: REAL; arScrew[98].rWidth : REAL; arScrew[98].rAngle_knives : REAL; arScrew[98].rMidle_line : REAL; arScrew[98].rInstal_support : REAL; arScrew[98].rPosX0 : REAL; arScrew[98].rPosX1 : REAL; arScrew[98].rPosX2 : REAL; arScrew[98].equip.place : WSTRING(10); arScrew[98].equip.name : WSTRING(20); arScrew[98].name : WSTRING(20); arScrew[99].rRstmax : REAL; arScrew[99].rRstmin : REAL; arScrew[99].iCountCycle : INT; arScrew[99].iActuatorsMove : INT; arScrew[99].iActuatorsStep : INT; arScrew[99].iActuatorsStartPos[0] : INT; arScrew[99].iActuatorsStartPos[1] : INT; arScrew[99].support[0].bPosition : BOOL; arScrew[99].support[0].arLength[0] : INT; arScrew[99].support[0].arLength[1] : INT; arScrew[99].support[0].name : WSTRING(20); arScrew[99].support[1].bPosition : BOOL; arScrew[99].support[1].arLength[0] : INT; arScrew[99].support[1].arLength[1] : INT; arScrew[99].support[1].name : WSTRING(20); arScrew[99].bDirRotate : BOOL; arScrew[99].rOut_diam : REAL; arScrew[99].rInner_diam : REAL; arScrew[99].rTurn_step : REAL; arScrew[99].rWidth : REAL; arScrew[99].rAngle_knives : REAL; arScrew[99].rMidle_line : REAL; arScrew[99].rInstal_support : REAL; arScrew[99].rPosX0 : REAL; arScrew[99].rPosX1 : REAL; arScrew[99].rPosX2 : REAL; arScrew[99].equip.place : WSTRING(10); arScrew[99].equip.name : WSTRING(20); arScrew[99].name : WSTRING(20); arScrew[100].rRstmax : REAL; arScrew[100].rRstmin : REAL; arScrew[100].iCountCycle : INT; arScrew[100].iActuatorsMove : INT; arScrew[100].iActuatorsStep : INT; arScrew[100].iActuatorsStartPos[0] : INT; arScrew[100].iActuatorsStartPos[1] : INT; arScrew[100].support[0].bPosition : BOOL; arScrew[100].support[0].arLength[0] : INT; arScrew[100].support[0].arLength[1] : INT; arScrew[100].support[0].name : WSTRING(20); arScrew[100].support[1].bPosition : BOOL; arScrew[100].support[1].arLength[0] : INT; arScrew[100].support[1].arLength[1] : INT; arScrew[100].support[1].name : WSTRING(20); arScrew[100].bDirRotate : BOOL; arScrew[100].rOut_diam : REAL; arScrew[100].rInner_diam : REAL; arScrew[100].rTurn_step : REAL; arScrew[100].rWidth : REAL; arScrew[100].rAngle_knives : REAL; arScrew[100].rMidle_line : REAL; arScrew[100].rInstal_support : REAL; arScrew[100].rPosX0 : REAL; arScrew[100].rPosX1 : REAL; arScrew[100].rPosX2 : REAL; arScrew[100].equip.place : WSTRING(10); arScrew[100].equip.name : WSTRING(20); arScrew[100].name : WSTRING(20)
      global variables Global_Variables
      Vizualization/
        TextList/
          text list OnOffList
          text list MbBoud
          text list NoYes
          text list ModeSysList
          text list typeEquip
          text list Direction
          text list MbParity
          text list MbStopbit
          text list TypeSetup
          text list DirectRotation
        image pool Images
        visualisation Waiting
        ImagesPool/
          image pool sensPool
          image pool PumpPool
          image pool ValvePool
        7_inch/
          visualisation _Actuators
          visualisation _SettingsEquipment
          visualisation _Diag_geomtry_rec
          visualisation _Support
          visualisation _Equipment_2
          visualisation _Equipment_3
          visualisation _Diag_WARNING
          visualisation _TypeMachine
          visualisation _Diag_support_rec
          visualisation _Equip_7inch
          visualisation _Equipment_4
          visualisation _Diag_save
          visualisation _Equipment_1
          visualisation _Diag_geomtry_work
          visualisation _Steel_7inch
          visualisation _SettingsSens_7inch
          visualisation _Alarms_7inch
          visualisation _MAIN_7inch
          visualisation _Equipment
          visualisation _Recipe_7inch
          visualisation _Diag_ok
          visualisation _SettingsActuators
          visualisation _Diag_equip
          visualisation _SettingsMain_7inch
          visualisation _TimeSetup_7inch
          visualisation _Diag_supKey
      Alarm Configuration
        alarm group AlarmGroup
            8 [Error]: Comparison Equal, ExpressionToCompare    TRUE, Expression Actuators.bDr1_error - "Ошибка драйвера актуатора 1"
            9 [Error]: Comparison Equal, ExpressionToCompare TRUE, Expression Actuators.bDr2_error - "Ошибка драйвера актуатора 2"
            1 [Error]: Comparison Equal, ExpressionToCompare TRUE, Expression Main.fbKkMotor.bOUT - "Сработало тепловое реле элекродвигателя маслостанции"
            3 [Error]: Comparison Equal, ExpressionToCompare TRUE, Expression Main.fbControl.bAlarm - "Ошибка дижения рабочего цилиндра"
            4 [Error]: Comparison Equal, ExpressionToCompare TRUE, Expression Main.fbTimeMotor.bService - "Проведите плановое плановое ТО"
            5 [Error]: Comparison Equal, ExpressionToCompare TRUE, Expression Main.bSnsH - "Достигнута максимально крайняя точка движения (координата X4)"
            6 [Error]: Comparison Equal, ExpressionToCompare TRUE, Expression Main.bSnsL - "Достигнута минимально крайняя точка движения (координата X3)"
            7 [Error]: Comparison Equal, ExpressionToCompare TRUE, Expression Main.bNoConnect - "Нет сигнала с модулем ПР"
        alarm group WarningGroup
            0 [Warning]: Comparison Equal, ExpressionToCompare TRUE, Expression warn.bStartPos - "Начальная позиция актуаторов выходит за допустимы предел"
            1 [Warning]: Comparison Equal, ExpressionToCompare TRUE, Expression warn.bMaxMove - "Расчитанных ход актуаторов больше, чем их возможный"
            2 [Warning]: Comparison Equal, ExpressionToCompare TRUE, Expression warn.bNotSupport - "Нет подходящей поддержки"
        AlarmStorage
        alarm class Error (priority 10, acknowledge REP)
        text list AlarmGroup
        text list WarningGroup
        alarm class Warning (priority 11, acknowledge REP)
    Debug : Debug, Production association OWEN, version 3.5.17.3001 (disabled)
        unmapped channels: RAM used, RAM free, Open files, Processor usage, Core temp, Enable Debug, Debug pause
    Info : Info, Production association OWEN, version 3.5.17.3001 (disabled)
        unmapped channels: VENDOR, DEVICE, SERIAL, RUNTIME, FIRMWARE, LINUX, TARGET, PROJECT, AUTHOR, VERSION, PROFILE, LASTCHANGES
    OwenRTC : OwenRTC, Production association OWEN, version 3.5.17.3001 (disabled)
        unmapped channels: Year, Month, Day, Hour, Minute, Second, Day of Week, Week of Year, Format Date, Format Time, UTC Offset, NTP Enabled, NTP Error, System Timer, Date And Time, Operating Time, New Year, New Month, New Day, New Hour, New Minute, New Second, New UTC Offset, Set Settings DT, Enable NTP, Prefer Server
    OwenCloud : OwenCloud, Production association OWEN, version 3.5.17.3001 (disabled)
        unmapped channels: OwenCloud enabled, Folder error, Symbol error, No Symbol Config, Status, Enable OwenCloud
    Buzzer : Buzzer, Production association OWEN, version 3.5.17.3001 (disabled)
        unmapped channels: Buzzer enabled, Enable Buzzer, Sound frequency
    Watchdog : Watchdog, Production association OWEN, version 3.5.17.3001 (disabled)
        unmapped channels: Exception Handling, Last Exception Code, Last Exception Description, Last Exception Time, Hardware Watchdog Flag, Power Reboot Count, Watchdog Reboot Count, Exception Reboot Count, Command Reboot Count, Reboot, Reset Counters
    Drives : Drives, Production association OWEN, version 3.5.17.3001 (disabled)
        unmapped channels: FS size, FS used, FS free, USB Mounted, USB Unmount done, USB size, USB used, USB free, MMC Mounted, MMC Unmount done, MMC size, MMC used, MMC free, FS wear, Enable Drives, USB Unmount, MMC Unmount
    Screen : Screen, Production association OWEN, version 3.5.17.3001 (disabled)
        unmapped channels: Get Brightness, Dim time, Off time, Full brightness, Dim brightness, Off brightness, Dim visu name, Off visu name, On visu name, Wake up
    Network : Network, Production association OWEN, version 3.5.17.3001 (disabled)
        unmapped channels: DHCP enabled, IP, Mask, Gateway, MAC, Hostname, Enable DHCP, New IP, New Mask, New Gateway, New Hostname, Set Settings
    Modbus_COM : Modbus COM, 3S - Smart Software Solutions GmbH, version 3.5.16.0
        settings: DataBits = 8; StopBits = 1; ComPort = 1
      Modbus_Master_COM_Port : Modbus Master, COM Port, 3S - Smart Software Solutions GmbH, version 3.5.17.0
          settings: Transmission = 'RTU'; ResponseTimeout = 50; TimeBetweenFrames = 30; Auto-restart communication = TRUE
        AI_module : Modbus Slave, COM Port, 3S - Smart Software Solutions GmbH, version 3.5.16.0
            settings: SlaveAddress = 16; ResponseTimeout = 20; UseExtendedFunctionCodes = TRUE; Channel 0.Function Code = 3; Channel 0.Read Offset = 16#0200; Channel 0.Read Length = 7; Channel 0.Write Offset = 0; Channel 0.Write Length = 0; Channel 0.Cycle Time = 20; Channel 1.Function Code = 16; Channel 1.Read Offset = 0; Channel 1.Read Length = 0; Channel 1.Write Offset = 16#0214; Channel 1.Write Length = 11; Channel 1.Cycle Time = 20; Channel 3.Function Code = 16; Channel 3.Read Offset = 0; Channel 3.Read Length = 0; Channel 3.Write Offset = 16#021F; Channel 3.Write Length = 4; Channel 3.Cycle Time = 20; Channel 4.Function Code = 3; Channel 4.Read Offset = 16#0207; Channel 4.Read Length = 3; Channel 4.Write Offset = 0; Channel 4.Write Length = 0; Channel 4.Cycle Time = 20
            input  inArWord : ARRAY[0..6] OF WORD  // Channel 0
            input  readSec : WORD  // Channel 0.Channel 0
            input  DI1 : WORD  // Channel 0.Channel 0
            input  DO1 : WORD  // Channel 0.Channel 0
            output writeX0 : WORD  // Channel 1.Channel 1
            output writeX1 : WORD  // Channel 1.Channel 1
            output writeX2 : WORD  // Channel 1.Channel 1
            output writeX3 : WORD  // Channel 1.Channel 1
            output writeX4 : WORD  // Channel 1.Channel 1
            output writeSec : WORD  // Channel 1.Channel 1
            output writeMode : WORD  // Channel 1.Channel 1
            output writeData : WORD  // Channel 1.Channel 1
            output writeMinL : WORD  // Channel 1.Channel 1
            output writeMaxL : WORD  // Channel 1.Channel 1
            output writeOffset : WORD  // Channel 1.Channel 1
            output writeImpMaxDr1 : WORD  // Channel 3.Channel 3
            output writeImpMaxDr2 : WORD  // Channel 3.Channel 3
            output writeImpSetpDr1 : WORD  // Channel 3.Channel 3
            output writeImpSetpDr2 : WORD  // Channel 3.Channel 3
            input  readStateDr : WORD  // Channel 4.Channel 4
            input  readCntImpDr1 : WORD  // Channel 4.Channel 4
            input  readCntImpDr2 : WORD  // Channel 4.Channel 4
            unmapped channels: Channel 1, Channel 3, Channel 4
  5ce3da45-db07-42e7-a21c-a00fff4ed8f6|D:\png для cWeb\KSp_alarm.png
  5ce3da45-db07-42e7-a21c-a00fff4ed8f6|D:\png для cWeb\SU_on.png
  5ce3da45-db07-42e7-a21c-a00fff4ed8f6|D:\png для cWeb\SU_off.png
  5ce3da45-db07-42e7-a21c-a00fff4ed8f6|background.jpeg
  5ce3da45-db07-42e7-a21c-a00fff4ed8f6|D:\png для cWeb\TO_SPAD.png
  5ce3da45-db07-42e7-a21c-a00fff4ed8f6|D:\png для cWeb\FO_alarm.png
  5ce3da45-db07-42e7-a21c-a00fff4ed8f6|background1.jpg
  5ce3da45-db07-42e7-a21c-a00fff4ed8f6|C:\Users\Андрей\Downloads\background_SuUP.jpg
  5ce3da45-db07-42e7-a21c-a00fff4ed8f6|C:\Users\Андрей\Downloads\лого1.png
  5ce3da45-db07-42e7-a21c-a00fff4ed8f6|C:\Users\Андрей\Downloads\background_FoDW.jpg
  5ce3da45-db07-42e7-a21c-a00fff4ed8f6|D:\png для cWeb\EK_on.png
  5ce3da45-db07-42e7-a21c-a00fff4ed8f6|C:\Users\Андрей\Downloads\miniLogo_white.png
  5ce3da45-db07-42e7-a21c-a00fff4ed8f6|C:\Users\Андрей\Downloads\background_FanUP.jpg
  5ce3da45-db07-42e7-a21c-a00fff4ed8f6|D:\png для cWeb\TO_freeze.png
  5ce3da45-db07-42e7-a21c-a00fff4ed8f6|D:\png для cWeb\DumpIn_off_op.png
  5ce3da45-db07-42e7-a21c-a00fff4ed8f6|D:\png для cWeb\EK_alarm.png
  5ce3da45-db07-42e7-a21c-a00fff4ed8f6|D:\png для cWeb\Pump_left_alarm.png
  5ce3da45-db07-42e7-a21c-a00fff4ed8f6|D:\png для cWeb\Fan_right_on.png
  5ce3da45-db07-42e7-a21c-a00fff4ed8f6|C:\Users\Андрей\Downloads\background_GenUP.jpg
  5ce3da45-db07-42e7-a21c-a00fff4ed8f6|D:\png для cWeb\SU_alarm.png
  5ce3da45-db07-42e7-a21c-a00fff4ed8f6|C:\Users\Андрей\Downloads\background_SuDW.jpg
  5ce3da45-db07-42e7-a21c-a00fff4ed8f6|D:\Program's\картинки для мнемосхем\svg\Arrow_Black_Left.svg
  5ce3da45-db07-42e7-a21c-a00fff4ed8f6|D:\png для cWeb\Filter_Alarm.png
  5ce3da45-db07-42e7-a21c-a00fff4ed8f6|D:\png для cWeb\KSp_off.png
  5ce3da45-db07-42e7-a21c-a00fff4ed8f6|D:\Program's\картинки для мнемосхем\Избранные\Warning.png
  5ce3da45-db07-42e7-a21c-a00fff4ed8f6|D:\png для cWeb\miniLOGO.png
  5ce3da45-db07-42e7-a21c-a00fff4ed8f6|D:\Program's\картинки для мнемосхем\png для cWeb\Filter.png
  5ce3da45-db07-42e7-a21c-a00fff4ed8f6|D:\png для cWeb\TO_on.png
  5ce3da45-db07-42e7-a21c-a00fff4ed8f6|D:\png для cWeb\circle_orange.png
  5ce3da45-db07-42e7-a21c-a00fff4ed8f6|D:\png для cWeb\circle_blue.png
  5ce3da45-db07-42e7-a21c-a00fff4ed8f6|C:\Users\Андрей\Downloads\background_FanDW.jpg
  5ce3da45-db07-42e7-a21c-a00fff4ed8f6|C:\Users\Андрей\Downloads\fon2.jpg
  5ce3da45-db07-42e7-a21c-a00fff4ed8f6|D:\png для cWeb\FO_off.png
  5ce3da45-db07-42e7-a21c-a00fff4ed8f6|D:\Program's\картинки для мнемосхем\svg\изначальные\WaterHot_right.svg
  5ce3da45-db07-42e7-a21c-a00fff4ed8f6|C:\Users\Андрей\Downloads\fon.jpg
  5ce3da45-db07-42e7-a21c-a00fff4ed8f6|C:\Users\Андрей\Downloads\background_KpUP.jpg
  5ce3da45-db07-42e7-a21c-a00fff4ed8f6|C:\Users\Андрей\Downloads\glyphicons-447-floppy-save@3x.png
  5ce3da45-db07-42e7-a21c-a00fff4ed8f6|D:\png для cWeb\Fan_right_off.png
  5ce3da45-db07-42e7-a21c-a00fff4ed8f6|D:\png для cWeb\Fan_right_off_alarm.png
  5ce3da45-db07-42e7-a21c-a00fff4ed8f6|D:\Program's\картинки для мнемосхем\svg\Arrow_Black_Right.svg
  5ce3da45-db07-42e7-a21c-a00fff4ed8f6|D:\png для cWeb\JTU.png
  5ce3da45-db07-42e7-a21c-a00fff4ed8f6|D:\png для cWeb\FO_Start.png
  5ce3da45-db07-42e7-a21c-a00fff4ed8f6|D:\png для cWeb\EK_off_alarm.png
  5ce3da45-db07-42e7-a21c-a00fff4ed8f6|D:\png для cWeb\Alarm.png
  5ce3da45-db07-42e7-a21c-a00fff4ed8f6|C:\Users\Андрей\Downloads\background_GenDW.jpg
  5ce3da45-db07-42e7-a21c-a00fff4ed8f6|D:\png для cWeb\KSp_on.png
  5ce3da45-db07-42e7-a21c-a00fff4ed8f6|D:\png для cWeb\Valve4.png
  5ce3da45-db07-42e7-a21c-a00fff4ed8f6|iconSave.png
  5ce3da45-db07-42e7-a21c-a00fff4ed8f6|D:\png для cWeb\DumpIn_off_middle.png
  5ce3da45-db07-42e7-a21c-a00fff4ed8f6|C:\Users\Андрей\Downloads\background_KpDW.jpg
  5ce3da45-db07-42e7-a21c-a00fff4ed8f6|D:\png для cWeb\circle.png
  5ce3da45-db07-42e7-a21c-a00fff4ed8f6|D:\png для cWeb\Fan_right_work.png
  5ce3da45-db07-42e7-a21c-a00fff4ed8f6|D:\png для cWeb\DumpIn_alarm.png
  5ce3da45-db07-42e7-a21c-a00fff4ed8f6|D:\png для cWeb\TO_off.png
  5ce3da45-db07-42e7-a21c-a00fff4ed8f6|D:\png для cWeb\DumpIn_off.png
  5ce3da45-db07-42e7-a21c-a00fff4ed8f6|diagram15.png
  5ce3da45-db07-42e7-a21c-a00fff4ed8f6|D:\png для cWeb\Valve1.png
  5ce3da45-db07-42e7-a21c-a00fff4ed8f6|D:\png для cWeb\Filter_Normal.png
  5ce3da45-db07-42e7-a21c-a00fff4ed8f6|C:\Users\Андрей\Downloads\logo.png
  5ce3da45-db07-42e7-a21c-a00fff4ed8f6|D:\png для cWeb\EK_on_alarm.png
  5ce3da45-db07-42e7-a21c-a00fff4ed8f6|D:\png для cWeb\Fan_right_on_alarm.png
  text list GlobalTextList
  5ce3da45-db07-42e7-a21c-a00fff4ed8f6|D:\png для cWeb\circle_yellow.png
  5ce3da45-db07-42e7-a21c-a00fff4ed8f6|D:\png для cWeb\Pump_left_off.png
  5ce3da45-db07-42e7-a21c-a00fff4ed8f6|C:\Users\Андрей\Downloads\background_MainUP.jpg
  5ce3da45-db07-42e7-a21c-a00fff4ed8f6|D:\png для cWeb\circle_light_blue.png
  5ce3da45-db07-42e7-a21c-a00fff4ed8f6|D:\Program's\картинки для мнемосхем\svg\Arrow_Black_Up.svg
  5ce3da45-db07-42e7-a21c-a00fff4ed8f6|D:\png для cWeb\Valve3.png
  5ce3da45-db07-42e7-a21c-a00fff4ed8f6|D:\png для cWeb\JTU_frost.png
  5ce3da45-db07-42e7-a21c-a00fff4ed8f6|лого.PNG
  5ce3da45-db07-42e7-a21c-a00fff4ed8f6|D:\png для cWeb\TO_alarm.png
  5ce3da45-db07-42e7-a21c-a00fff4ed8f6|D:\png для cWeb\JTU_alarm.png
  5ce3da45-db07-42e7-a21c-a00fff4ed8f6|D:\png для cWeb\Valve0.png
  5ce3da45-db07-42e7-a21c-a00fff4ed8f6|C:\Users\Андрей\Downloads\background_FoUP.jpg
  5ce3da45-db07-42e7-a21c-a00fff4ed8f6|C:\Users\Андрей\Downloads\background_ToDW.jpg
  5ce3da45-db07-42e7-a21c-a00fff4ed8f6|C:\Users\Андрей\Downloads\background_ToUP.jpg
  5ce3da45-db07-42e7-a21c-a00fff4ed8f6|D:\png для cWeb\Filter.png
  5ce3da45-db07-42e7-a21c-a00fff4ed8f6|D:\png для cWeb\DumpIn_on.png
  5ce3da45-db07-42e7-a21c-a00fff4ed8f6|diagram16.png
  5ce3da45-db07-42e7-a21c-a00fff4ed8f6|D:\png для cWeb\Pump_left_Work.png
  5ce3da45-db07-42e7-a21c-a00fff4ed8f6|D:\png для cWeb\FO_work.png
  5ce3da45-db07-42e7-a21c-a00fff4ed8f6|C:\Users\Андрей\Downloads\лого.png
  5ce3da45-db07-42e7-a21c-a00fff4ed8f6|D:\png для cWeb\TO_work.png
  5ce3da45-db07-42e7-a21c-a00fff4ed8f6|C:\Users\Андрей\Downloads\background_MainDW.jpg
  5ce3da45-db07-42e7-a21c-a00fff4ed8f6|D:\png для cWeb\Pump_left_on_alarm.png
  5ce3da45-db07-42e7-a21c-a00fff4ed8f6|D:\png для cWeb\EK_off.png
  5ce3da45-db07-42e7-a21c-a00fff4ed8f6|D:\Program's\картинки для мнемосхем\svg\Arrow_Black_Down.svg
  5ce3da45-db07-42e7-a21c-a00fff4ed8f6|D:\png для cWeb\JTU_on.png
  5ce3da45-db07-42e7-a21c-a00fff4ed8f6|D:\png для cWeb\circle_green.png
  5ce3da45-db07-42e7-a21c-a00fff4ed8f6|D:\png для cWeb\DumpIn_off_cl.png
  GlobalImagePool
  5ce3da45-db07-42e7-a21c-a00fff4ed8f6|D:\png для cWeb\circle_red.png
  5ce3da45-db07-42e7-a21c-a00fff4ed8f6|D:\png для cWeb\Pump_left_on.png
*)

// Device/Application/POUs/gp/Data_types/warning
TYPE warning :
STRUCT
	 bGeneral 		:BOOL;
	 bNotSupport	:BOOL; //нет подходящего кронштейна
	 bStartPos	:BOOL; //начальная точка заходит за возможные пределы дв. актуаторов
	 bMaxMove		:BOOL; //расчетная длина движения актуаторов больше чем возможные пределы
END_STRUCT
END_TYPE

// Device/Application/POUs/gp/Data_types/recType
TYPE recType EXTENDS dataBase:
STRUCT
	rOut_diam	: REAL:=0.0;//Наружный диаметр D2
	rInner_diam	: REAL:=0.0;//Внутренний диаметр D1
	rTurn_step	: REAL:=0.0;//Шаг витка L
	rWidth		: REAL:=0.0;//толщина заготовки
	rAngle_knives	: REAL:=0.0;//Угол наклона ножей Ω
	rMidle_line		: REAL:=0.0;//Положение средней линии, ФАКТ
	rInstal_support	: REAL:=0.0;//Установка поддержки, ФАКТ	
	rPosX0 			:REAL:=0.0; //начало координаты отсчета цикла
	rPosX1 			:REAL:=0.0; //Обратный ход гидроцилиндра от Х2 до Х1
	rPosX2 			:REAL:=0.0; //задание на выдвижение гидроцилиндра до Х2
	equip			: equipment;//оснастка станка
END_STRUCT
END_TYPE

// Device/Application/POUs/gp/Data_types/SupportType
TYPE SupportType EXTENDS dataBase :
STRUCT
	arLength 	:ARRAY [0..1] OF INT;//длина опоры [0]-длина L  [1]-длина для  Г
END_STRUCT
END_TYPE

// Device/Application/POUs/gp/Data_types/Ustav
TYPE Ustav :
STRUCT
		rMaxPoint :REAL := 230.0; //макс допустимая длина  x4
		rMinPoint :REAL := 150.0; //мин допустимая длина x3

		rAccuracy :REAL :=0.7;//погрешность,мм
		iTimeMoveEr :INT := 1;//аварийное время на проверку движения		
		iTimeService :INT := 100;//время сревисного обслуж, ч
		
		rMaxLength  :REAL := 250.0;//макс длина измерения датчика
		rMinLength  :REAL := 0.0;//мин. длина измерения датчика
		rOffset :REAL := 0.0;//коррекция датчика перемещения

		rInitAngleSupport :REAL := 45.0;//начальный угол установки опоры для калькулятора
		
		bEnAutoMatrix :BOOL; //Станок с автоматической матрицей, версия ПРО 
		iHeightMatrix  :INT:=624;//Высота матрицы, для версии ПРО станка
		iMaxActuatorsMove	:INT:=180; //максимальный ход актуаторов, для версии ПРО станка
		iMaxImpDr1 : INT:= 1000;//максимальное допустимо кол-во имп для дв1, для версии ПРО станка
		iMaxImpDr2 : INT:= 1000;//максимальное допустимо кол-во имп для дв2, для версии ПРО станка
END_STRUCT
END_TYPE

// Device/Application/POUs/gp/Data_types/test
TYPE test :
STRUCT
	distance	:REAL;
	startCycle	: ARRAY[0..1] OF UINT;
	endCycle	:ARRAY[0..1] OF UINT;
END_STRUCT
END_TYPE

// Device/Application/POUs/gp/Data_types/Union_Real
TYPE Union_Real :
UNION
	rVal:REAL;
	wWord: ARRAY[0..1] OF WORD;
END_UNION
END_TYPE

// Device/Application/POUs/gp/Data_types/dataBase
TYPE dataBase :
STRUCT
		name: WSTRING(20):="";//наименование
END_STRUCT
END_TYPE

// Device/Application/POUs/gp/Data_types/OperTime
//структура времени наработки, сеанс и общее
TYPE OperTime :
STRUCT
	dwTimeTotal			:	DWORD;(*Общее время наработки , в мин.*)
	
	dwHourTotal			:	DWORD;(*Время наработки , часы.*)
	dwMinTotal			:	DWORD;(*Время наработки , минуты.*)
	dwHourSeans			:	DWORD;(*Сеансовое время наработки , часы.*)
	dwMinSeans			:	DWORD;(*Сеансовое время наработки , минуты.*)

	dwLastServ	:	DWORD;//время последнего ТО
END_STRUCT
END_TYPE

// Device/Application/POUs/gp/Data_types/FindOfEq
TYPE FindOfEq :
STRUCT
	find: Equipment;
	bestFind:Equipment;
END_STRUCT
END_TYPE

// Device/Application/POUs/gp/Data_types/recType2
TYPE recType2 EXTENDS recType :
STRUCT
	 rRstmax 	 :REAL;//Наружный радиус заготовки, Rstmax(для конусных витков)
	 rRstmin 	 :REAL;//Наружный радиус заготовки, Rstmin(для конусных витков)
	 iCountCycle :INT;//Примерное количество циклов(для конусных витков)
	 iActuatorsMove :INT; //Ход актуаторов  (для конусных витков)
	 iActuatorsStep :INT; //Смещение актуаторов в цикле  (для конусных витков)
	 iActuatorsStartPos :ARRAY [0..1]  OF INT;//начальная позиция актуаторов (для конусных витков)		 
	 support :ARRAY [0..1]  OF	SupportType2;//установленые опоры  (для конусных витков)
	 bDirRotate :BOOL;//направление вращение заготовки 0-правый 1-левый

END_STRUCT
END_TYPE

// Device/Application/POUs/gp/Data_types/Equipment
TYPE Equipment EXTENDS dataBase :
STRUCT
	place: WSTRING(10):="";//стелаж, ряд, ячейка
END_STRUCT
END_TYPE

// Device/Application/POUs/gp/Data_types/middle_line
TYPE middle_line :
STRUCT
	val:	UINT;
	valMin: UINT;
	valMax: UINT;
END_STRUCT
END_TYPE

// Device/Application/POUs/gp/Data_types/Steel
TYPE Steel EXTENDS dataBase:
STRUCT
	t:DINT;//предел текучести
END_STRUCT
END_TYPE

// Device/Application/POUs/gp/Data_types/Accept_struct
TYPE Accept_struct :
STRUCT
	bX0 	: BOOL;// принять точку старта x0
	bX1  	: BOOL; //принять точки x1
	bX2  	: BOOL; //принять точки x2	
	bAct 	: BOOL; //принять данные для актуатора
	bSup 	: BOOL; //принять данные кронштейна	
	bRec	: BOOL; //принять данные рецепта	
END_STRUCT
END_TYPE

// Device/Application/POUs/gp/Data_types/SupportType2
TYPE SupportType2 EXTENDS SupportType:
STRUCT
	bPosition 	:BOOL; //положение опоры 0 - L(Pos1), 1 -Г(Pos2)
END_STRUCT
END_TYPE

// Device/Application/Global_Variables
VAR_GLOBAL RETAIN
	SP		 			: Ustav;
	operTimeMotor		: OperTime;
	
END_VAR

VAR_GLOBAL 
	arScrew :ARRAY[0..SIZE_SCREWS] OF RecType2;
	arEquip :ARRAY [0..SIZE_EQUIPS] OF Equipment;
	arSteel :ARRAY [0..SIZE_STEELS] OF Steel;	
	arSupports :ARRAY [0..SIZE_SUPPORT] OF SupportType;
	
	sRecGroupName :STRING:='RecGroup';  // Имя выбранной группы рецептов
	sRecName :STRING:='Rec'; 
	sRecGroupName1 :STRING:='SteelGroup';  // Имя выбранной группы рецептов
	sRecName1 :STRING:='Steel'; 
	sRecGroupName2 :STRING:='EquipGroup';  // Имя выбранной группы рецептов
	sRecName2 :STRING:='Equip'; 
	sRecGroupName3 :STRING:='SupGroup';  // Имя выбранной группы рецептов
	sRecName3 :STRING:='Support'; 	
	
	bGoCalc :BOOL:=FALSE;//кнопка "пересчитать" шнек
	bActiveViewRec :BOOL:=FALSE;//Активно меню Рецептов

	warn : warning;
		
	bLogin		: BOOL;	//флаг что доступ открыт
	bReset		: BOOL;	//кнопка сброса аварии	
	bResetTO 	: BOOL;
	bResetOP	: BOOL;
	curPoint 	: recType2;
	setPoint 	: recType2;
	
	btnAccept : Accept_struct;
	
	iMode 	  	: INT; //0-непрерывный, 1-цикличный, 2-ручной(установка х0) ,3-проверка точности
	bPedalFrd	: BOOL;//педаль 1 движение вперед;
	bPedalRev	: BOOL;//педаль 2 движение назад;
	bKkMotor 	: BOOL;//тепловое реле двигателя
	bEmStop  	: BOOL;//Аварийный останов
	bBut_OnOff  : BOOL;//кнопка вкл. откл маслостанции
	bBut_Off: BOOL;//кнопкаоткл маслостанции
	bOnMotor	: BOOL;//пуск мотора маслостанции
	bOnValveFrd	: BOOL;//вкл. клапан н дв вперед
	bOnValveRev	: BOOL;//вкл. клапан н дв назад
END_VAR

VAR_GLOBAL CONSTANT
	SIZE_STEELS  :INT:=100;
	SIZE_EQUIPS  :INT:=100;
	SIZE_SCREWS  :INT:=100;
	SIZE_SUPPORT :INT:=100;
END_VAR

// Device/Application/POUs/gp/Main
PROGRAM Main
VAR
	fbEmergencyStop :MESSAGEEX;
	fbKkMotor :MESSAGEEX;
	fbDelay :TON;

	fbTimeMotor: OPERATING_TIME_V1;	
	fbControl : fbControl_sys;

	bErrLamp : BOOL; //лампа ошибки
	bNoConnect: BOOL;//ошибка связи с ПР100
	
	bSnsH		: BOOL:=FALSE;	//ошибка верхнего предела
	bSnsL		: BOOL:=FALSE;	//ошибка нижнего предела
	memReadSec 	: WORD:=0; //сохранные секунды часов реального времени

	AI_val		: Union_REAL;
	snsLenght	: Union_REAL;
	MeXH		: MessageEx;
	MeXL		: MessageEx;
	
	FirstCycle :BOOL:=TRUE;
	
	fbSimMove 	: simulateMove;
	tp_bGoCalc :tp;
END_VAR

IF FirstCycle THEN
	CalcTech.rAngle_support :=sp.rInitAngleSupport;
	FirstCycle:=FALSE;
END_IF

Visu_var();

IF bActiveViewRec THEN
	recipes();
END_IF

tp_bGoCalc(In:=bGoCalc, pt:=T#1S);//костылина для проходки нескольких циклов
IF tp_bGoCalc.Q THEN
	CalcTech();
END_IF

//лампа авария	
	fbEmergencyStop(
		bDI:= NOT bEmStop, 
		bEnbl:= TRUE, 
		bLock:= TRUE, 
		iDelEn:= 0, 
		bReset:= bReset, 
		bOUT=> );
		
	fbKkMotor(
		bDI:= NOT bKkMotor, 
		bEnbl:= TRUE, 
		bLock:= FALSE, 
		iDelEn:= 1, 
		bReset:= bReset, 
		bOUT=> );

	MeXH(bDI:=FALSE,
		bEnbl:= snsLenght.rVal >= sp.rMaxPoint,
		bLock:= FALSE,
		iDelEn:=0,
		bReset:=bReset ,
		bOUT=> bSnsH);
		
	MeXL(bDI:=FALSE,
		bEnbl:= snsLenght.rVal <= sp.rMinPoint,
		bLock:= FALSE ,
		iDelEn:=0,
		bReset:=bReset ,
		bOUT=> bSnsL);

		
	
	bErrLamp := fbEmergencyStop.bOUT OR fbKkMotor.bOUT OR fbControl.bAlarm;
//	наработка
	fbTimeMotor(bEn:= bOnMotor, 
				iTimeTO:= sp.iTimeService, 
				bResetTO:= bResetTO, 
				bReset:= bResetOP, 
				op:= operTimeMotor, 
				bService=> );

// 
fbControl(rCurLength:= snsLenght.rVal, 
				setX:= setPoint, 
				recX:= recipes.Screw, 
				rAccuracy:= sp.rAccuracy, 
				bMoveFrd:= bOnValveFrd, 
				bMoveRev:= bOnValveRev, 
				bReset:= bReset , 
				iTimeErr:= sp.iTimeMoveEr, 
				Accept:= btnAccept, 
				rLengthFromX0=> , 
				curX=> curPoint, 
				bAlarm=> );		

//
IF btnAccept.bRec THEN
	setPoint :=recipes.Screw;
END_IF

//				
IF 	btnAccept.bX0 OR  btnAccept.bX1 OR  btnAccept.bX2 OR bGoCalc THEN
		btnAccept.bX0:=  btnAccept.bX1 := btnAccept.bX2 :=bGoCalc :=FALSE;
END_IF

//
IF sp.bEnAutoMatrix THEN
	Actuators(bDirRotate := curPoint.bDirRotate,//направление вращение заготовки
				iCycleNumb := curPoint.iCountCycle,//число циклов
				iCalcStep := curPoint.iActuatorsStep,//шаг смещения
				iStartPos := curPoint.iActuatorsStartPos,//начальная поз. акт)
				Support	:= curPoint.support	);
END_IF
	
	
ACT_INPUT();

ACTION ACT_INPUT:
//Входы выходы 
	bPedalFrd	:= DI1.0 ;//педаль 1 движение вперед;
	bPedalRev	:= DI1.1 ;//педаль 2 движение назад;
	bKkMotor := DI1.2;//тепловое реле двигателя
	bEmStop  := DI1.3;//Аварийный останов
	bBut_OnOff  := DI1.4;//кнопка вкл. откл маслостанции\
	bBut_Off := DI1.5;//доп кнопка откл.маслостанции
	
	bOnValveFrd := DO1.0;//вкл. клапан н дв вперед
	bOnMotor := DO1.1;//пуск мотора маслостанции
	bOnValveRev := DO1.2;//вкл. клапан н дв назад

	
//Сигнал AI
	AI_val.wWord[0]:=inArWord[3];
	AI_val.wWord[1]:=inArWord[4];
	snsLenght.wWord[0]:=inArWord[5];
	snsLenght.wWord[1]:=inArWord[6];
	
//сетевые данные 
	writeX0	:= REAL_TO_WORD(fbControl.curX.rPosX0*10);
	writeX1 := REAL_TO_WORD(fbControl.rCalcX1*10);
	writeX2 := REAL_TO_WORD(fbControl.rCalcX2*10);
	writeX3 := REAL_TO_WORD(sp.rMinPoint*10);
	writeX4	:= REAL_TO_WORD(sp.rMaxPoint*10);
	writeMode:= INT_TO_WORD(iMode);
	writeData.0 := bErrLamp;	// остановка маслостанции
	
	writeMinL := REAL_TO_WORD(sp.rMinLength*10);
	writeMaxL := REAL_TO_WORD(sp.rMaxLength*10);
	writeOffset := REAL_TO_WORD(sp.rOffset*10);

	fbDelay(in:= NOT fbDelay.Q, pt:=T#2S);
	
	IF fbDelay.Q THEN
		bNoConnect := memReadSec <> readSec;
		memReadSec := readSec;
	END_IF
	
	whatTime(uiSec=>writeSec);
END_ACTION

END_PROGRAM

// Device/Application/POUs/gp/CalcTech
PROGRAM CalcTech
 VAR 
 //геометрия заготовки
	 rWidth_turn:REAL;//Ширина витка	
	 rSmaller_radius:REAL;// Меньший радиус  R1.1 для ACT_ANGLE_MACHINE()
	 rLarge_radius:REAL;// Больший радиус   R2.1 для ACT_ANGLE_MACHINE()
	 
	 rOut_radius: REAL;//Вх. наружный диаметр R2
	 rInner_radius: REAL;//Вх. внутренний диаметр R1
	 rPercA1_1: REAL; //Процентное отношение А1.1
	 rPercA2_1: REAL; //Процентное отношение А2.1
	 
	 x,y,ks,L7,M7,M6 :LREAL;
	 rWidthCutoutSmall:REAL;//Ширина выреза меньшая
	 rWidthCutoutLarge:REAL;//Ширина выреза большая
	 rAngleCutout:REAL;//Угол раскрытия выреза
	 rKdp : REAL;//выбранный коэффициент
	 rKfact: REAL;//Коэффициент поправки
	 rS1: REAL;//Толщина S1
	 rAngeY1_1, rAngeY2_2 : REAL; //Угол γ1.1 γ2.2
	 
	 i : INT;

//угол установки
  	rTrapezoidHeight :REAL; //высота трапеции для ACT_ELASTIC_MOVE()
	rTrapezoidWidth :REAL; //ширина трапеции для ACT_ELASTIC_MOVE()
	rSideA1: REAL;//Сторона	A1 относительно оси заготовки
	rSideA2: REAL;//Сторона	A2 относительно оси заготовки
	rSideA1_1: REAL;//Сторона	A1 относительно оси трубы для ACT_GEOMetry()
	rSideA2_1: REAL;//Сторона	A1 относительно оси трубы для ACT_GEOMetry()
	rPercA1: REAL; //Процентное отношение rSideA1
	rPercA2: REAL; //Процентное отношение rSideA2
	rMidLine: REAL; //Положение средней линии R3
	rAngle_y1: REAL;//Угол γ1
	rAngle_y2: REAL;//Угол	γ2
	rAngle_y: REAL;//Угол γ для ACT_GEOMetry()
	rAngle_y1_1: REAL;//Угол	γ1.1
	rAngle_y2_1: REAL;//Угол	γ2.1
	dX2: REAL;//Остаточная деформация ΔХ2
    X2x2: REAL;//Параметр рабочего хода Х2х2
	
	rCathetC : REAL;//Катет c
	rInstal_support: REAL;

//упругие перемещения
	rBd:REAL;//отношение b/d;
	rCoefK1:REAL; // коэффиценты соотношений К1 
	rCoefK3:REAL; // коэффиценты соотношений К3 	
	rLimElastic:REAL;//Предел текучести при сдвиге
 
	rElasticAnge:REAL;//Упругая составляющая угла закручивания, град
	rMoveKnife:REAL;//Перемещение ножей соответствующие углу, мм
	rElasticOffset:REAL;  //Поправка на упругость	Z1 для ACT_ANGLE_MACHINE()
	
//автоматические матрицы
	rSupLenghtMin :REAL; //минимальная длина кронштейна 
	rRoutmax	:REAL:=225.0;  //Радиус наружный максимальный (для конусных витков)
	rRoutmin	:REAL:=155.0;  //Радиус наружный минимальный (для конусных витков)
	rRins: REAL:=108;//Внутренний радиус, Rins (для конусных витков)
	rLeftSupMaxMove : REAL;//Установка Rstmax, левая поддержка
	rLeftSupMinMove : REAL;//Установка Rstmin, левая поддержка
	rRightSupMaxMove : REAL;//Установка Rstmax, правая поддержка
	rRightSupMinMove : REAL;//Установка Rstmin, правая поддержка
END_VAR

VAR_INPUT
	 rOut_diam: REAL:=505;//вх. наружный диаметр D2 или диаметр наружный максимальный (для конусных витков)
	 rInner_diam: REAL:=108;//вх. внутренний диаметр D1 или Внутренний диаметр (для конусных витков)
	 rTurn_step: REAL:=100;//вх. шаг витка L
	 rWidth: REAL:=3;//вх. толщина заготовки
	 rCount_turn: REAL:=200;//вх. количество витков
		 
	 bDirection:BOOL:=TRUE;//вх. направление витка 1-правый 0-левый 
	 bStrengthened:BOOL:=FALSE;//вх. 1-усиленный 0-нет
	 steel :steel:=(name:="09Г2С", t:= 450);//вх. марка стали
	 rAngle_support :REAL:=45;//вх. угол установленной опоры
	 
	 rCoef_KL:REAL:=0.0;//вх. Поправкана срабатывание соленоидов
	
 //Автоматическая матрица 
	bEnConicalScrew :BOOL; //вх. включить режим расчета для КОНУСНЫЙх шнеков 
	rOut_diamMin :REAL:=400.0; //вх. диаметр наружный минимальный (для конусных витков)
	rRotationCircle :REAL:=360;//вх. поворот окружности витка, S (для конусных витков)
	bDirRotation	:BOOL:=FALSE;//вх. направление навивки витка 0-правый 1-левый 
	
END_VAR

VAR_OUTPUT
 //work piece Параметры заготовки 
	 rWpOut_diam	 : REAL;//вых.наружный диаметр
	 rWpInner_diam	 : REAL;//вых.внутренний диаметр
	 rWpRebordHeight : REAL;//вых высота реборды
	 rWpAngle		 : REAL;//вых угол раскрытия выреза
	 // rCoef:REAL;//Выбранный коэффициент
	 
 //Параметры настройки станка  Machine Settings
	 rMsInstal_support : REAL;//вых. установка поддержки
	 rMsFactInstal_support : REAL;//вых. установка поддержки, ФАКТ для спиральных ножей
	 rMsMidle_line 		   : REAL;//вых. положение средней линии, ГЕОМ
	 rMsFactMidle_line 		: REAL;//вых. положение ср. линии, ФАКТ для спиральных ножей
	 rMsAngle_knives :REAL;//вых. угол наклона ножей Ω
	 rMsX2		:REAL;//вых. параметр рабочего хода Х2;
	 msEquipment	: findofEq;//вых. необходимая маркировка оснастки	 
	 
	 dataForRec : RecType2;
 //Автоматическая матрица
	 rRstmax 	 :REAL;//вых.наружный радиус заготовки, Rstmax(для конусных витков)
	 rRstmin 	 :REAL;//вых.наружный радиус заготовки, Rstmin(для конусных витков)
	 rRstins 	 :REAL;//вых.внутренний радиус заготовки, Rstins(для конусных витков)
	 iCountCycle :INT;//вых.примерное количество циклов(для конусных витков)
	 rActuatorsMove :REAL; //вых. ход актуаторов  (для конусных витков)
	 rActuatorsStep :REAL; //вых. смещение актуаторов в цикле  (для конусных витков)
	 support :ARRAY [0..1] OF SupportType2;//вых.установленая опора  (для конусных витков)
	 iStartSupPos :ARRAY [0..1] OF INT;//вых.начальная позиция актуаторов (для конусных витков)	

END_VAR

VAR CONSTANT
	//таблица коэффициентов для расчета геометрии
	arCoefData : ARRAY [0..11,0..1] OF REAL:= [	0.00065, 1.2,
												0.00070, 1.3,
												0.00075, 1.35,
												0.00080, 1.4,
												0.001, 1.5,
												0.0025, 1.6,
												0.00415, 1.7,
												0.0055, 1.8,
												0.0085, 1.9,
												0.01, 2,
												0.0125, 2.2];
												
	//таблица коэффициентов для расчета упругих перемещений	(Коэффициенты соотношений K1,K3))										
	arCoefDataK1 : ARRAY [0..9,0..2] OF REAL:= [
											10, 0.333, 0.333,
											8, 0.313, 0.313,
											6, 0.299, 0.299,
											4.5, 0.283, 0.28,
											3, 0.267, 0.263,
											2.5, 0.258, 0.249,
											2, 0.246, 0.229,
											1.75, 0.239, 0.214,
											1.5, 0.231, 0.156,
											1, 208, 141];	

	PI:REAL:=3.14159265;
	DENSITY: DINT:=7860; //плотность
	G:DINT:=80000;//модуль юнга, сдвига
	
END_VAR

rInner_radius := rRins;

CalcTech.rOut_diam := rRoutmax * 2;
CalcTech.rInner_diam := rRins *2;
CalcTech.rOut_diamMin := rRoutmin *2;

IF bEnConicalScrew THEN
	rOut_radius := (rRoutmax + rRoutmin)/2;
ELSE
	rOut_radius := rRoutmax;
END_IF

rWidth_turn :=(rOut_radius-rInner_radius);

ACT_GEOMETRY();
ACT_ANGLE_MACHINE();

rMsFactInstal_support := rMsInstal_support-(rMsMidle_line-rMsFactMidle_line);

msEquipment := fcFindOfEquip(
			rMidLine:= rMsFactMidle_line, //средняя линия
			rRebordHeight:= rWpRebordHeight, //высота реборды
			rAngle:=rMsAngle_knives , //угол
			bStrengthened:= bStrengthened, // усилинный
			bDirection:= bDirection, //направление
			db:= ADR(arEquip), //массив блок данных
			lengthDb:= 100 //размер массива
		);
		
IF sp.bEnAutoMatrix THEN
	IF bEnConicalScrew THEN
		ACT_AUTO_MATRIX();
	ELSE
		ACT_MATRIX();
	END_IF		
END_IF	

//dataForRec.name - записывается через диалог
dataForRec.rOut_diam := rOut_radius * 2;
dataForRec.rInner_diam := rInner_radius * 2;
dataForRec.rTurn_step :=rTurn_step;
dataForRec.rWidth :=rWidth;

dataForRec.rAngle_knives:=rMsAngle_knives;
dataForRec.rMidle_line:= rMsFactMidle_line;
dataForRec.rInstal_support:= rMsFactInstal_support;

IF msEquipment.find.name = "нет совпадений" THEN
	dataForRec.equip:=msEquipment.bestFind;
ELSE
	dataForRec.equip:=msEquipment.find;
END_IF
	
dataForRec.rPosX0:= 0;
dataForRec.rPosX1:= 15;
dataForRec.rPosX2:= rMsX2;

 dataForRec.rRstmax :=	rRstmax;//Наружный радиус заготовки, Rstmax(для конусных витков)
 dataForRec.rRstmin :=	rRstmin;//Наружный радиус заготовки, Rstmin(для конусных витков)
 dataForRec.iCountCycle := iCountCycle;//Примерное количество циклов(для конусных витков)
 dataForRec.iActuatorsMove := REAL_TO_INT(rActuatorsMove); //Ход актуаторов  (для конусных витков)
 dataForRec.iActuatorsStep := REAL_TO_INT(rActuatorsStep); //Смещение актуаторов в цикле  (для конусных витков)
 dataForRec.support := support;//установленые опоры  (для конусных витков)
 dataForRec.iActuatorsStartPos :=	iStartSupPos;//начальная позиция актуаторов (для конусных витков)

METHOD PRIVATE remap : UINT
VAR_INPUT
	indx:UINT;//индекс массива
	remapArr:POINTER TO UINT;//шаблонный массив для переназначения 
	lengthRemapArr:UINT; //размер массива
	valueArr:POINTER TO middle_line;
	originalValue:UINT ;// округленное вх значение
	
	remapOffset:UINT;//дополнительное смещение индекса
END_VAR
    IF (indx = 0 OR lengthRemapArr <= indx OR remapArr[indx] = 0)  THEN
      remap:= originalValue ;
	ELSE
	  remap:= valueArr[remapArr[indx]+remapOffset].val  ;
	END_IF
END_METHOD

METHOD PRIVATE roundTo : REAL
VAR_INPUT
END_VAR
END_METHOD

// Converts from degrees to radians.
METHOD PRIVATE DEGR_TO_RAD : REAL 
VAR_INPUT
	degrees :REAL;
END_VAR
DEGR_TO_RAD := (degrees * 3.1415926535) / 180;
END_METHOD

METHOD PRIVATE fcFindOfEquip : FindOfEq;//расчет поиск оснастки

VAR_INPUT
	rMidLine :REAL;//вх значение расчетной средней линии
	rRebordHeight :REAL;//вх Высота реборды
	rAngle:REAL;//вх угол
	bStrengthened:BOOL;//вх. 1-усиленный 0-нет
	bDirection:BOOL;//вх. направление 1-правый 0-левый
	db : POINTER TO Equipment;//массив с библ. данными
	lengthDb :INT;//длина массива с библ. данными
END_VAR

VAR
	iMidLine :UINT; //округленное вх значение расчетной средней линии
	iRebordHeight :UINT;//округленное вх Высота реборды
	iAngle:UINT;//округленное вх угол опоры
	
	iIndxML:UINT;//найденый индекс в массиве ML 
	iIndxCH:UINT;//найденый индекс в массиве CH 
	iLnB1,iLnB2,iLnB3,iLnB4,iLnB5 :UINT;
	iRb1, iRb2, iRb3, iRb4 :UINT;
	prefix:WSTRING;
	
	iIndxAngle:UINT;//найденый индекс в массиве ANGLE_VAL 
	iAngleB1, iAngleB2 :UINT;
	
	opts:ARRAY[0..30] OF WSTRING;
	i,j: INT;
END_VAR

VAR CONSTANT
	//параметры средней линии
	 	ML: ARRAY [0..43] OF middle_line:=[ //
		(val:=15,valMin:=14,valMax:=19),
		(val:=20,valMin:=20,valMax:=24),
		(val:=25,valMin:=25,valMax:=29),
		(val:=30,valMin:=30,valMax:=34),
		(val:=35,valMin:=35,valMax:=39),
		(val:=40,valMin:=40,valMax:=44),
		(val:=45,valMin:=45,valMax:=49),
		(val:=50,valMin:=50,valMax:=53),
		(val:=55,valMin:=54,valMax:=57),
		(val:=60,valMin:=58,valMax:=65),
		(val:=70,valMin:=66,valMax:=75),
		(val:=80,valMin:=76,valMax:=85),
		(val:=90,valMin:=86,valMax:=95),
		(val:=100,valMin:=96,valMax:=105),
		(val:=110,valMin:=106,valMax:=115),
		(val:=120,valMin:=116,valMax:=125),
		(val:=130,valMin:=126,valMax:=135),
		(val:=140,valMin:=136,valMax:=145),
		(val:=150,valMin:=146,valMax:=155),
		(val:=160,valMin:=156,valMax:=165),
		(val:=170,valMin:=166,valMax:=175),
		(val:=180,valMin:=176,valMax:=190),
		(val:=200,valMin:=191,valMax:=210),
		(val:=220,valMin:=211,valMax:=235),
		(val:=250,valMin:=236,valMax:=260),
		(val:=270,valMin:=261,valMax:=285),
		(val:=300,valMin:=286,valMax:=315),
		(val:=320,valMin:=316,valMax:=335),
		(val:=350,valMin:=336,valMax:=360),
		(val:=370,valMin:=361,valMax:=385),
		(val:=400,valMin:=386,valMax:=415),
		(val:=420,valMin:=416,valMax:=435),
		(val:=450,valMin:=436,valMax:=460),
		(val:=470,valMin:=461,valMax:=485),
		(val:=500,valMin:=486,valMax:=515),
		(val:=520,valMin:=516,valMax:=535),
		(val:=550,valMin:=536,valMax:=560),
		(val:=570,valMin:=561,valMax:=585),
		(val:=600,valMin:=586,valMax:=615),
		(val:=620,valMin:=616,valMax:=635),
		(val:=650,valMin:=636,valMax:=660),
		(val:=670,valMin:=661,valMax:=685),
		(val:=700,valMin:=686,valMax:=715),
		(val:=720,valMin:=716,valMax:=735)];

 	//Выбор средней линии В1
	REMAP_ML1:ARRAY [0..42] OF UINT:= [0, 1, 2, 3, 4, 5, 6, 7,  8,  9,  10, 11, 12, 13, 14, 15, 16, 17, 18, 19, 20, 21, 22, 23, 24, 25, 26, 27, 28, 29, 30, 31, 32, 33, 34, 35, 36, 37, 38, 39, 40, 41, 42];
    //Выбор средней линии В2
	REMAP_ML2:ARRAY [0..43] OF UINT:= [0, 0, 1, 2, 3, 4, 5, 6,  7,  8,  9,  10, 11, 12, 13, 14, 15, 16, 17, 18, 19, 20, 21, 22, 23, 24, 25, 26, 27, 28, 29, 30, 31, 32, 33, 34, 35, 36, 37, 38, 39, 40, 41, 42];
	//Выбор средней линии В3
	REMAP_ML3:ARRAY [0..42] OF UINT:= [1, 2, 3, 4, 5, 6, 7, 8,  9,  10, 11, 12, 13, 14, 15, 16, 17, 18, 19, 20, 21, 22, 23, 24, 25, 26, 27, 28, 29, 30, 31, 32, 33, 34, 35, 36, 37, 38, 39, 40, 41, 42, 43];
  	//Выбор средней линии В4
	REMAP_ML4:ARRAY [0..41] OF UINT:=[2, 3, 4, 5, 6, 7, 8, 9,  10, 11, 12, 13, 14, 15, 16, 17, 18, 19, 20, 21, 21, 22, 23, 24, 25, 26, 27, 28, 29, 30, 31, 32, 33, 34, 35, 36, 37, 38, 39, 40, 41, 42];
  	//Выбор средней линии В5
	REMAP_ML5:ARRAY [0..42] OF UINT:= [3, 4, 5, 6, 7, 8, 9, 10, 11, 12, 13, 14, 15, 16, 17, 18, 19, 20, 20, 21, 21, 22, 23, 24, 25, 26, 27, 28, 29, 30, 31, 32, 33, 34, 35, 36, 37, 38, 39, 40, 41, 42, 43];

	//высота ножа
 	CUTTER_HEIGHT :ARRAY [0..24] OF UINT:=[ 0, 30,50,80,100,120,150,170,200,220,250,300,350,400,450,500,550,600,650,700,750,800,850,900,950 ];
	REMAP_CH2 :ARRAY [0..21] OF UINT:= [1, 2, 3, 4, 5, 6, 7, 8,  9,  10, 11, 12, 13, 14, 15, 16, 17, 18, 19, 20, 21, 22];
	REMAP_CH3 :ARRAY [0..21] OF UINT:= [2, 3, 4, 5, 6, 7, 8, 9,  10, 11, 12, 13, 14, 15, 16, 17, 18, 19, 20, 21, 22, 22];
	REMAP_CH4 :ARRAY [0..22] OF UINT:= [3, 4, 5, 6, 7, 8, 9, 10, 11, 12, 13, 14, 15, 16, 17, 18, 19, 20, 21, 22, 0, 22, 22];

	//угол
	ANGLE_VAL:ARRAY [0..12]OF UINT:= [0,4,6,8,10,12,14,15,16,17,18,19,20];
	
	nothing :Equipment:= (name:="нет совпадений", place:="");
	
END_VAR
rRebordHeight:=rRebordHeight+5;//костыль какой то хз зачем

iMidLine := REAL_TO_UINT(rMidLine);//округление  
iRebordHeight := REAL_TO_UINT(rRebordHeight);//округление 

iIndxML := pickRangeNumber(iMidLine, ADR(ML), 43);//найденый индекс в массиве ML 

iLnB1 := remap(iIndxML, ADR(REMAP_ML1), 42, ADR(ML), iMidLine,0,);
iLnB2 := remap(iIndxML, ADR(REMAP_ML2), 43, ADR(ML), iMidLine,0);
iLnB3 := remap(iIndxML, ADR(REMAP_ML3), 42, ADR(ML), iMidLine,0);
iLnB4 := remap(iIndxML, ADR(REMAP_ML4), 41, ADR(ML), iMidLine,0);
iLnB5 := remap(iIndxML, ADR(REMAP_ML5), 42, ADR(ML), iMidLine,0);

iIndxCH := pickRangeNumberLinear(iRebordHeight, ADR(CUTTER_HEIGHT), 24);

IF iIndxCH = 0 THEN
	iRb1 := iRebordHeight;
	iRb2 := iRebordHeight;
	iRb3 := iRebordHeight;
	iRb4 := iRebordHeight;
ELSE	
	iRb1 := CUTTER_HEIGHT[iIndxCH+1];		
	iRb2 := remap_1(iIndxCH, ADR(REMAP_CH2), 21, ADR(CUTTER_HEIGHT), iRebordHeight,1);	
	iRb3 := remap_1(iIndxCH, ADR(REMAP_CH3), 21, ADR(CUTTER_HEIGHT), iRebordHeight,1);	
	iRb4 := remap_1(iIndxCH, ADR(REMAP_CH4), 21, ADR(CUTTER_HEIGHT), iRebordHeight,1);		
END_IF

prefix :=wconcat(wconcat( wconcat(SEL(bDirection, "L", "R"), "-"),  SEL(bStrengthened, "N" , "S")), "-");

iAngle:= REAL_TO_UINT(rAngle);
iIndxAngle := pickRangeNumberLinear(iAngle, ADR(ANGLE_VAL), 12);

IF iIndxAngle = 0 THEN
	iAngleB1 := ceil(rAngle);
	iAngleB2 := iAngleB1 + iAngle;
ELSE
	iAngleB1 := ANGLE_VAL[iIndxAngle+1];
	iAngleB2 := ANGLE_VAL[MIN(10,iIndxAngle+2)];
END_IF

opts[0] := wconcat( prefix, wconcat( UINT_TO_WSTRING(iRb1), wconcat( "-", wconcat( UINT_TO_WSTRING(iAngleB1) , wconcat("-",  UINT_TO_WSTRING(iLnB1) ) ) ) ) );
opts[1] := wconcat( prefix, wconcat( UINT_TO_WSTRING(iRb2), wconcat( "-", wconcat( UINT_TO_WSTRING(iAngleB1) , wconcat("-",  UINT_TO_WSTRING(iLnB1)) ) ) ) );
opts[2] := wconcat( prefix, wconcat( UINT_TO_WSTRING(iRb3), wconcat( "-", wconcat( UINT_TO_WSTRING(iAngleB1) , wconcat("-",  UINT_TO_WSTRING(iLnB1)) ) ) ) );
opts[3] := wconcat( prefix, wconcat( UINT_TO_WSTRING(iRb1), wconcat( "-", wconcat( UINT_TO_WSTRING(iAngleB2) , wconcat("-",  UINT_TO_WSTRING(iLnB1)) ) ) ) );   
opts[4] := wconcat( prefix, wconcat( UINT_TO_WSTRING(iRb2), wconcat( "-", wconcat( UINT_TO_WSTRING(iAngleB2) , wconcat("-",  UINT_TO_WSTRING(iLnB1)) ) ) ) );   
opts[5] := wconcat( prefix, wconcat( UINT_TO_WSTRING(iRb3), wconcat( "-", wconcat( UINT_TO_WSTRING(iAngleB2) , wconcat("-",  UINT_TO_WSTRING(iLnB1)) ) ) ) ); 
opts[6] := wconcat( prefix, wconcat( UINT_TO_WSTRING(iRb3), wconcat( "-", wconcat( UINT_TO_WSTRING(iAngleB1) , wconcat("-",  UINT_TO_WSTRING(iLnB2)) ) ) ) ); 
opts[7] := wconcat( prefix, wconcat( UINT_TO_WSTRING(iRb3), wconcat( "-", wconcat( UINT_TO_WSTRING(iAngleB1) , wconcat("-",  UINT_TO_WSTRING(iLnB3)) ) ) ) ); 	
opts[8] := wconcat( prefix, wconcat( UINT_TO_WSTRING(iRb2), wconcat( "-", wconcat( UINT_TO_WSTRING(iAngleB1) , wconcat("-",  UINT_TO_WSTRING(iLnB2)) ) ) ) ); 	
opts[9] := wconcat( prefix, wconcat( UINT_TO_WSTRING(iRb2), wconcat( "-", wconcat( UINT_TO_WSTRING(iAngleB1) , wconcat("-",  UINT_TO_WSTRING(iLnB3)) ) ) ) ); 

opts[10] := wconcat( prefix, wconcat( UINT_TO_WSTRING(iRb3), wconcat( "-", wconcat( UINT_TO_WSTRING(iAngleB2) , wconcat("-",  UINT_TO_WSTRING(iLnB2) ) ) ) ) );
opts[11] := wconcat( prefix, wconcat( UINT_TO_WSTRING(iRb3), wconcat( "-", wconcat( UINT_TO_WSTRING(iAngleB2) , wconcat("-",  UINT_TO_WSTRING(iLnB3) ) ) ) ) ); 
opts[12] := wconcat( prefix, wconcat( UINT_TO_WSTRING(iRb2), wconcat( "-", wconcat( UINT_TO_WSTRING(iAngleB2) , wconcat("-",  UINT_TO_WSTRING(iLnB2) ) ) ) ) ); 
opts[13] := wconcat( prefix, wconcat( UINT_TO_WSTRING(iRb2), wconcat( "-", wconcat( UINT_TO_WSTRING(iAngleB2) , wconcat("-",  UINT_TO_WSTRING(iLnB3) ) ) ) ) ); 
opts[14] := wconcat( "П-Н-", wconcat( UINT_TO_WSTRING(iRb3), wconcat( "-", wconcat( UINT_TO_WSTRING(iAngleB1) , wconcat("-",  UINT_TO_WSTRING(iLnB4) ) ) ) ) ); 
opts[15] := wconcat( prefix, wconcat( UINT_TO_WSTRING(iRb3), wconcat( "-", wconcat( UINT_TO_WSTRING(iAngleB1) , wconcat("-",  UINT_TO_WSTRING(iLnB4) ) ) ) ) ); 
opts[16] := wconcat( prefix, wconcat( UINT_TO_WSTRING(iRb3), wconcat( "-", wconcat( UINT_TO_WSTRING(iAngleB2) , wconcat("-",  UINT_TO_WSTRING(iLnB4) ) ) ) ) ); 
opts[17] := wconcat( prefix, wconcat( UINT_TO_WSTRING(iRb4), wconcat( "-", wconcat( UINT_TO_WSTRING(iAngleB1) , wconcat("-",  UINT_TO_WSTRING(iLnB4) ) ) ) ) ); 
opts[18] := wconcat( prefix, wconcat( UINT_TO_WSTRING(iRb4), wconcat( "-", wconcat( UINT_TO_WSTRING(iAngleB2) , wconcat("-",  UINT_TO_WSTRING(iLnB4) ) ) ) ) ); 
opts[19] := wconcat( prefix, wconcat( UINT_TO_WSTRING(iRb4), wconcat( "-", wconcat( UINT_TO_WSTRING(iAngleB1) , wconcat("-",  UINT_TO_WSTRING(iLnB5) ) ) ) ) ); 

opts[20] := wconcat( prefix, wconcat( UINT_TO_WSTRING(iRb4), wconcat( "-", wconcat( UINT_TO_WSTRING(iAngleB2) , wconcat("-",  UINT_TO_WSTRING(iLnB5) ) ) ) ) ); 
opts[21] := wconcat( prefix, wconcat( UINT_TO_WSTRING(iRb4), wconcat( "-", wconcat( UINT_TO_WSTRING(iAngleB1) , wconcat("-",  UINT_TO_WSTRING(iLnB1) ) ) ) ) );     
opts[23] := wconcat( prefix, wconcat( UINT_TO_WSTRING(iRb4), wconcat( "-", wconcat( UINT_TO_WSTRING(iAngleB2) , wconcat("-",  UINT_TO_WSTRING(iLnB1) ) ) ) ) );   
opts[24] := wconcat( prefix, wconcat( UINT_TO_WSTRING(iRb4), wconcat( "-", wconcat( UINT_TO_WSTRING(iAngleB1) , wconcat("-",  UINT_TO_WSTRING(iLnB3) ) ) ) ) );         
opts[25] := wconcat( prefix, wconcat( UINT_TO_WSTRING(iRb4), wconcat( "-", wconcat( UINT_TO_WSTRING(iAngleB1) , wconcat("-",  UINT_TO_WSTRING(iLnB2) ) ) ) ) );   
opts[26] := wconcat( prefix, wconcat( UINT_TO_WSTRING(iRb1), wconcat( "-", wconcat( UINT_TO_WSTRING(iAngleB1) , wconcat("-",  UINT_TO_WSTRING(iLnB2) ) ) ) ) );   
opts[27] := wconcat( prefix, wconcat( UINT_TO_WSTRING(iRb1), wconcat( "-", wconcat( UINT_TO_WSTRING(iAngleB1) , wconcat("-",  UINT_TO_WSTRING(iLnB3) ) ) ) ) );        
opts[28] := wconcat( prefix, wconcat( UINT_TO_WSTRING(iRb1), wconcat( "-", wconcat( UINT_TO_WSTRING(iAngleB1) , wconcat("-",  UINT_TO_WSTRING(iLnB3) ) ) ) ) );   
opts[29] := wconcat( prefix, wconcat( UINT_TO_WSTRING(iRb1), wconcat( "-", wconcat( UINT_TO_WSTRING(iAngleB2) , wconcat("-",  UINT_TO_WSTRING(iLnB3) ) ) ) ) );      
opts[30] := wconcat( prefix, wconcat( UINT_TO_WSTRING(iRb1), wconcat( "-", wconcat( UINT_TO_WSTRING(iAngleB2) , wconcat("-",  UINT_TO_WSTRING(iLnB2) ) ) ) ) );    
    
FOR i:=0 TO 30 DO   
	FOR j:=0 TO lengthDb DO  
		IF (db[j].name<>"") AND (db[j].name = opts[i]) THEN
			fcFindOfEquip.find.name := db[j].name;
			fcFindOfEquip.find.place := db[j].place;
			fcFindOfEquip.bestFind.name:=opts[0];
			RETURN;
		END_IF
	END_FOR
END_FOR  

fcFindOfEquip.find := nothing;
fcFindOfEquip.bestFind.name:=opts[0];
END_METHOD

METHOD PRIVATE fcFindOfSup : bool//
VAR_INPUT
	maxMotion :INT;//ход актуаторов макс
	minMotion :INT;//ход актуаторов мин
	arr	:POINTER TO SupportType;//каталог опор
	length : INT;//размер массива

END_VAR
VAR
	i,j: INT;
	maxPos, minPos :INT;
END_VAR
VAR_OUTPUT
	result : SupportType2;
	strPos : INT; //стартовые позиции
END_VAR
FOR	i:=0 TO 1 DO
	FOR	j:=0 TO length DO
		
		IF arr[j].name = "" THEN
			CONTINUE	;
		END_IF
		
		//для поз 
		maxPos := arr[j].arLength[i] + sp.iHeightMatrix;
		minPos := arr[j].arLength[i] + (sp.iHeightMatrix - sp.iMaxActuatorsMove);
	
		IF maxPos >= maxMotion AND minPos <= minMotion THEN
			result.name := arr[j].name;
			result.bPosition := INT_TO_BOOL(i);
			result.arLength := arr[j].arLength;
			
			//strPos := minMotion-minPos-arr[j].arLength[i];
			strPos := sp.iHeightMatrix+arr[j].arLength[i]-minMotion;
			
			fcFindOfSup := 1; //удачно
			
			RETURN;
		END_IF
		
	END_FOR
END_FOR	

fcFindOfSup := 0; //нет подходящего кронштейна
END_METHOD

METHOD PRIVATE remap_1 : UINT
VAR_INPUT
	indx:UINT;//индекс массива
	remapArr:POINTER TO UINT;//шаблонный массив для переназначения 
	lengthRemapArr:UINT; //размер массива
	valueArr:POINTER TO UINT;
	originalValue:UINT ;// округленное вх значение
	
	remapOffset:UINT;//дополнительное смещение индекса
END_VAR
    IF (indx = 0 OR lengthRemapArr <= indx OR remapArr[indx] = 0)  THEN
      remap_1:= originalValue ;
	ELSE
	  remap_1:= valueArr[remapArr[indx]+remapOffset]  ;
	END_IF
END_METHOD

 // Converts from radians to degrees.
METHOD PRIVATE RAD_TO_DEGR : REAL
VAR_INPUT
	radians :REAL;
END_VAR
RAD_TO_DEGR := (radians *180) / 3.1415926535;
END_METHOD

ACTION ACT_AUTO_MATRIX:
(*вариант из ексель*)
	rRstins  := rSmaller_radius;//Внутренний радиус заготовки, Rstins
	rRstmax := rRoutmax - rRins + rRstins;//Наружный радиус заготовки, Rstmax
	rRstmin := rRoutmin - rRins + rRstins;//Наружный радиус заготовки, Rstmin
	
	iCountCycle := REAL_TO_INT(15/(360/rRotationCircle));//Примерное количество циклов 
	rActuatorsMove := (rRstmax-rRstmin)-(rRstmax-rRstmin)*rAngle_support/rRotationCircle;//макс ход актуаторов
	rActuatorsStep := rActuatorsMove/iCountCycle; //длина шага актуаторов.мм	
		
 	IF sp.iMaxActuatorsMove >= rActuatorsMove THEN

		IF bDirRotation THEN//в зависимости от на правления вращения заготовки
			rRightSupMaxMove :=rRstmax - (rRstmax-rRstmin) * rAngle_support/rRotationCircle;
			rLeftSupMaxMove :=  rRstmax;
			
			rRightSupMinMove := rRstmin;
			rLeftSupMinMove := rRstmin + (rRstmax-rRstmin) * rAngle_support/rRotationCircle;
		ELSE
			rLeftSupMaxMove:= rRstmax - (rRstmax-rRstmin) * rAngle_support/rRotationCircle;
			rRightSupMaxMove := rRstmax;
			
			rLeftSupMinMove	 := rRstmin;
			rRightSupMinMove := rRstmin + (rRstmax-rRstmin) * rAngle_support/rRotationCircle;
		END_IF

 		warn.bNotSupport := NOT fcFindOfSup(maxMotion:= REAL_TO_INT(rLeftSupMaxMove),minMotion:= REAL_TO_INT(rLeftSupMinMove), arr:= ADR(arSupports), length:= 100, result=>support[0], strPos =>iStartSupPos[0]); 
 		warn.bNotSupport := NOT fcFindOfSup(maxMotion:= REAL_TO_INT(rRightSupMaxMove),minMotion:= REAL_TO_INT(rRightSupMinMove), arr:= ADR(arSupports), length:= 100,  result=>support[1], strPos =>iStartSupPos[1]); 
 	ELSE
 		warn.bMaxMove :=TRUE;//расчетная длина движения актуаторов больше чем возможные пределы
 	END_IF
END_ACTION

METHOD PRIVATE pickRangeNumber : UINT //по вх. параметру выбор крайних значений и числа средней линии
VAR_INPUT
	x:UINT;
	arr	:POINTER TO middle_line;
	length: UINT;//размер массива
END_VAR

VAR
	i:UINT:=0;
END_VAR
FOR i:=0 TO length DO   
   IF arr[i].valMin <= x AND x <= arr[i+1].valMin THEN (*было  x <= arr[i+1].valMAX *)
      pickRangeNumber:= i;
		RETURN;
   END_IF
  
END_FOR
END_METHOD

ACTION ACT_GEOMETRY:
//из расчета угла установки
	rSideA1_1 := (rInner_radius*(SIN(DEGR_TO_RAD(rAngle_support/2))))*2;
	rSideA2_1 := (rOut_radius*(SIN(DEGR_TO_RAD(rAngle_support/2))))*2;
	
//из расчета геометрии
L7:= rCount_turn/8.0/4.0;
M7:= SQRT(EXPT(rSideA1_1,2)+EXPT((L7*2.0),2)) ;
M6:= SQRT(EXPT(rSideA2_1,2)+EXPT((L7*2.0),2)) ;

rPercA1_1 :=LREAL_TO_REAL( (M7*100)/(M7+M6) );
rPercA2_1 :=100-rPercA1_1;//

rAngeY1_1 := 90-(rAngle_y/100*rPercA2_1);
rAngeY2_2:= 90-(rAngle_y/100*rPercA1_1); 

	ks:= rOut_radius/rInner_radius/rTurn_step/rWidth;	//!!! rOut_diam, rInner_diam
	FOR i:=0 TO 10 DO 	
		IF ks < arCoefData[i,0] AND i=0 THEN
			rKdp:=arCoefData[i,1];
			
		ELSIF ks > arCoefData[i-1, 0] AND ks < arCoefData[i, 0] THEN
			rKdp:=arCoefData[i,1];
			
		ELSIF ks > arCoefData[10, 0] THEN
			rKdp:=2.5;	
		END_IF
		
	END_FOR
	rKfact := rOut_radius / rInner_radius/ rKdp; // !!!rOut_diam, rInner_diam
	
rS1:= ( SIN(DEGR_TO_RAD(rAngeY1_1))*rWidth )+( (rWidth -( SIN(DEGR_TO_RAD(rAngeY1_1))*rWidth)) / rKfact);
	
x :=  (SQRT(EXPT(pi,2)*EXPT((rInner_radius*2),2)+EXPT(rTurn_step,2)))*rS1 /rWidth ; // !!!rOut_diam, rInner_diam
y :=  SQRT(EXPT(pi,2)*EXPT((rOut_radius*2),2)+EXPT(rTurn_step,2)); // !!!rOut_diam, rInner_diam

rSmaller_radius := LREAL_TO_REAL( rWidth_turn* x / (y-x) );
rLarge_radius := rWidth_turn+rSmaller_radius;

rAngleCutout := LREAL_TO_REAL( 360.0*( (6.28*rLarge_radius-y)/(6.28*rLarge_radius) ) );
rWidthCutoutSmall := 2 * rSmaller_radius* SIN(DEGR_TO_RAD(rAngleCutout));
rWidthCutoutLarge := 2 * rLarge_radius* SIN(DEGR_TO_RAD(rAngleCutout)); 

rWpOut_diam :=2*rLarge_radius;
rWpInner_diam :=2*rSmaller_radius;	
rWpRebordHeight := (rWpOut_diam-rWpInner_diam)/2;
rWpAngle := rAngleCutout;
END_ACTION

METHOD PRIVATE pickRangeNumberLinear : UINT //выбор границ числа линии
VAR_INPUT
	x:UINT;
	arr	:POINTER TO UINT;
	length: UINT;//размер массива
END_VAR

VAR
	i:UINT:=0;
END_VAR
FOR i:=0 TO length DO   
   IF arr[i] <= x AND x <= arr[i+1] THEN 
      pickRangeNumberLinear:= i;
		RETURN;
   END_IF
  
END_FOR
END_METHOD

ACTION ACT_ANGLE_MACHINE:
rSideA1 := (rSmaller_radius*(SIN(DEGR_TO_RAD(rAngle_support/2))))*2;
rSideA2 := (rLarge_radius*(SIN(DEGR_TO_RAD(rAngle_support/2))))*2;

rPercA1 := (rSideA1/2*100)/((rSideA1+rSideA2)/2);
rPercA2 := 100- rPercA1;

rTrapezoidWidth := (rSideA1 +rSideA2)/2;
rTrapezoidHeight := (COS(DEGR_TO_RAD(rAngle_support/2))*(rWpRebordHeight/2))*2;

rMidLine := (rLarge_radius - rSmaller_radius)/2+rSmaller_radius;

rAngle_y1:= RAD_TO_DEGR(ATAN(rTurn_step/(2*rInner_radius*pi)));
rAngle_y2:= RAD_TO_DEGR(ATAN(rTurn_step/(2*rOut_radius*pi)));
rAngle_y := rAngle_y1-rAngle_y2;
rAngle_y1_1:= rAngle_y/100*rPercA2;
rAngle_y2_1:= rAngle_y/100*rPercA1;
	
dX2:=(TAN(DEGR_TO_RAD(rAngle_y2_1)))*(rSideA2/2);

ACT_ELASTIC_MOVE();
X2x2 := dX2*2+ rElasticOffset;//!!!!!!!

//выходные значения
rMsMidle_line := rMidLine;
IF bStrengthened THEN
	rMsFactMidle_line:= rMidLine-(8.5/TAN(DEGR_TO_RAD(rAngle_support/2)));
ELSE
		
	rMsFactMidle_line:= rMidLine-(5/TAN(DEGR_TO_RAD(rAngle_support/2)));
END_IF
rMsAngle_knives := RAD_TO_DEGR(ATAN(X2x2/2/(rLarge_radius - rMidLine)));

//
rCathetC := rWidth * COS(DEGR_TO_RAD(90-rMsAngle_knives));
rInstal_support := rLarge_radius + rCathetC;

//выходные значения
rMsInstal_support := rInstal_support + 100;
rMsX2:= X2x2-rCoef_KL;
END_ACTION

METHOD PRIVATE ceil : UINT//возвращает округленное число в большую сторону
VAR_INPUT
	rIn :REAL;
END_VAR

VAR
	iIn:UINT;
	
END_VAR
iIn := REAL_TO_UINT (rIn*10);

IF 0 <> (iIn MOD 10) THEN//если есть остатко то округляем в +1
	ceil := (iIn/10)+1;
ELSE
	ceil := REAL_TO_UINT(rIn);	
END_IF
END_METHOD

ACTION ACT_MATRIX:
(*вариант из ексель*)
	rRstins  := rSmaller_radius;//Внутренний радиус заготовки, Rstins
	rRstmax := rLarge_radius;//Наружный радиус заготовки, Rstmax
	rRstmin := rLarge_radius;//Наружный радиус заготовки, Rstmin

	iCountCycle := 0;//Примерное количество циклов 
	rActuatorsMove := 0.0;
	rActuatorsStep := 0.0; //длина шага актуаторов.мм	
 
	IF bDirRotation THEN//в зависимости от на правления вращения заготовки
			rRightSupMaxMove := rRstmax;
			rLeftSupMaxMove := rRstmax - (rRstmax-rRstmin) * rAngle_support/rRotationCircle;
			
			rRightSupMinMove := rRstmin - (rRstmax-rRstmin) * rAngle_support/rRotationCircle;
			rLeftSupMinMove := rRstmin;
	ELSE
			rRightSupMaxMove:= rRstmax - (rRstmax-rRstmin) * rAngle_support/rRotationCircle;
			rLeftSupMaxMove := rRstmax;
			
			rRightSupMinMove := rRstmin;
			rLeftSupMinMove := rRstmin - (rRstmax-rRstmin) * rAngle_support/rRotationCircle;
	END_IF

warn.bNotSupport := NOT fcFindOfSup(maxMotion:= REAL_TO_INT(rLeftSupMaxMove),minMotion:= REAL_TO_INT(rLeftSupMinMove), arr:= ADR(arSupports), length:= 100, result=>support[0], strPos =>iStartSupPos[0]); 
warn.bNotSupport := NOT fcFindOfSup(maxMotion:= REAL_TO_INT(rRightSupMaxMove),minMotion:= REAL_TO_INT(rRightSupMinMove), arr:= ADR(arSupports), length:= 100,  result=>support[1], strPos =>iStartSupPos[1]);
END_ACTION

ACTION ACT_ELASTIC_MOVE:
rBd := rTrapezoidHeight / rWidth;

	FOR i:=0 TO 9 DO 	
		IF rBd > arCoefDataK1[i,0] AND i=0 THEN
			rCoefK1:=arCoefDataK1[i,1];
			rCoefK3:=arCoefDataK1[i,2];
			
		ELSIF rBd > arCoefDataK1[i, 0] AND rBd < arCoefDataK1[i-1, 0] THEN
			rCoefK1:=arCoefDataK1[i,1];
			rCoefK3:= arCoefDataK1[i,2];
			
		ELSIF rBd < arCoefDataK1[9, 0] THEN
			rCoefK1:= 0.195;
			rCoefK3:= 0.12;
		END_IF
		
	END_FOR
	
rLimElastic := LREAL_TO_REAL((DINT_TO_REAL(steel.t)/SQRT(3.0)) );

rElasticAnge := RAD_TO_DEGR(rCoefK1/rCoefK3*(rLimElastic*rTrapezoidWidth/DINT_TO_REAL(G)/rWidth));
rMoveKnife := TAN(DEGR_TO_RAD(rElasticAnge))*rTrapezoidHeight;

rElasticOffset :=rMoveKnife/1.5;
END_ACTION

END_PROGRAM

// Device/Application/POUs/gp/Visu_var
PROGRAM Visu_var
VAR
	stValveFrd :STRING;
	stValveRev :STRING;	
	stMotor :STRING;
	stOperTimeSeans :STRING;
	stOperTimeTotal :STRING;
	
	ShowWaiting: VU.FbOpenDialog;
	point: VU.VisuStructPoint;
	exitWait: BOOL;
	DelayWait:TON;
END_VAR

IF bOnValveFrd THEN
	stValveFrd:='ValvePool.1';
ELSE
	stValveFrd:='ValvePool.0';
END_IF

IF bOnValveRev THEN
	stValveRev:='ValvePool.1';
ELSE
	stValveRev:='ValvePool.0';
END_IF

IF bOnMotor THEN
	stMotor:='PumpPool.1';
	
ELSIF	main.fbKkMotor.bOUT THEN
	stMotor:='PumpPool.2';
ELSE
	stMotor:='PumpPool.0';
END_IF

stOperTimeSeans := concat(concat(DWORD_TO_STRING(operTimeMotor.dwHourSeans), ':'), DWORD_TO_STRING(operTimeMotor.dwMinSeans));
stOperTimeTotal := concat(concat(DWORD_TO_STRING(operTimeMotor.dwHourTotal), ':'), DWORD_TO_STRING(operTimeMotor.dwMinTotal));

//окно ожидания
bLogin := visuElems.CurrentUserGroupId <> 0;//"None";

//
(*DelayWait(in:= NOT ( bLogin OR exitWait OR bPedalFrd OR bPedalRev), PT:=T#15S);
*)
warn.bGeneral := warn.bMaxMove OR warn.bNotSupport OR warn.bStartPos;
point.iX := 150;
point.iY := 100;
ShowWaiting(
	xExecute:= warn.bGeneral, 
	xDone=> , 
	xBusy=> , 
	xError=> , 
	itfClientFilter:= VU.Globals.AllClients, 
	eError=> , 
	sDialogName:= '_Diag_WARNING', 
	xModal:= TRUE, 
	pTopLeftPosition:= ADR(point));

IF bReset THEN
	 warn.bMaxMove := warn.bNotSupport := warn.bStartPos := FALSE;
END_IF

END_PROGRAM

// Device/Application/POUs/gp/recipes
PROGRAM recipes
VAR
	idxArScrew:INT;
	Screw:RecType2; 
	
	idxArEquip:INT;
	Equip:Equipment; 
	
	idxArSteel:INT;
	Steel:Steel;
	
	idxArSupport:INT;
	Support: SupportType;	
	
	i,j,k:INT:=0;
	commandRec :RecipeManCommands;
END_VAR

Support.name:= WCONCAT( WCONCAT("L", int_to_wstring(support.arLength[0])), WCONCAT(" - Г", int_to_wstring(support.arLength[1])) );

METHOD PUBLIC addData : BOOL
VAR_INPUT
	par:INT;
END_VAR
CASE par OF
	0:
		addData:=addScrew();
	1:
		addData:=addEquip();
	2:
		addData:=addSteel();
	3:
		addData:=addSupport();	
ELSE
	addData:=FALSE;
END_CASE
END_METHOD

METHOD DelData : BOOL
VAR_INPUT
	par:INT;
END_VAR
CASE par OF
	0:
		DelData:=DelScrew();
	1:
		DelData:=DelEquip();
	2:
		DelData:=DelSteel();
	3:
		DelData:=DelSupport();	
ELSE
	DelData:=FALSE;
END_CASE
END_METHOD

METHOD PUBLIC AddEquip : BOOL
VAR_INPUT
END_VAR
VAR
	i,idxFind:INT:=0;
	step:UINT;
END_VAR
step:=SIZEOF(equipment);

IF findName(ADR(arEquip),SIZE_SCREWS*step, step,Equip.name) THEN	
	AddEquip:=FALSE;
	RETURN;		
ELSE	
	FOR i:=0 TO SIZE_EQUIPS DO
		IF arEquip[i].name = "" THEN
			idxArEquip := i;
			arEquip[idxArEquip] := Equip;
			AddEquip :=TRUE;
			RETURN;
		END_IF	
	END_FOR
		AddEquip :=FALSE;

END_IF
END_METHOD

METHOD DelScrew : BOOL
VAR_INPUT
END_VAR
VAR
	i:int:=0;
END_VAR
VAR CONSTANT
	NOTHING :recType2:=(name:="",rOut_diam:=0.0,	rInner_diam:=0.0,rTurn_step:=0.0,rWidth:=0.0,rPosX0 :=0.0,rPosX1:=0.0,rPosX2 :=0.0);
END_VAR
FOR i:=idxArScrew TO SIZE_SCREWS DO 
	arScrew[i]:=arScrew[i+1];
	arScrew[i+1]:=NOTHING;
END_FOR
Screw := NOTHING;
DelScrew:=TRUE;
END_METHOD

METHOD DelSteel : BOOL
VAR_INPUT
END_VAR
VAR
	i:int:=0;
END_VAR
VAR CONSTANT
	NOTHING :Steel:=(name:="", t:=0);
END_VAR
FOR i:=idxArSteel TO SIZE_SteelS DO 
	arSteel[i]:=arSteel[i+1];
	arSteel[i+1]:=NOTHING;
END_FOR
Steel := NOTHING;
DelSteel:=TRUE;
END_METHOD

METHOD setScrew : BOOL
VAR_INPUT
END_VAR
	arScrew[idxArScrew]:= screw;
END_METHOD

METHOD PUBLIC AddScrew : BOOL
VAR_INPUT
END_VAR
VAR
	i,idxFind:INT:=0;
	step:UINT;
	search :BOOL;
END_VAR
step:=SIZEOF(recType);
search :=findName(ADR(arScrew), SIZE_SCREWS*step, step, Screw.name);

IF search THEN	
	AddScrew:=FALSE;
	RETURN;		
ELSE	
	FOR i:=0 TO SIZE_SCREWS DO
		IF arScrew[i].name = "" THEN
			idxArScrew := i;
			arScrew[idxArScrew] := screw;
			AddScrew :=TRUE;
			RETURN;
		END_IF	
	END_FOR
	AddScrew :=FALSE;
END_IF
END_METHOD

METHOD PUBLIC setData : BOOL
VAR_INPUT
	par:INT;
END_VAR
CASE par OF
	0:
		SetScrew();
	1:
		SetEquip();
	2:
		SetSteel();
	3:
		SetSupport();		
ELSE
	SetData:=FALSE;
END_CASE
END_METHOD

METHOD getSteel : BOOL
VAR_INPUT
END_VAR
	Steel := arSteel[idxArSteel] ;
END_METHOD

METHOD DelEquip : BOOL
VAR_INPUT
END_VAR
VAR
	i:int:=0;
END_VAR
VAR CONSTANT
	NOTHING :Equipment:=(name:="", place:="");
END_VAR
FOR i:=idxArEquip TO SIZE_EQUIPS DO 
	arEquip[i]:=arEquip[i+1];
	arEquip[i+1]:=NOTHING;
END_FOR
Equip := NOTHING;
DelEquip:=TRUE;
END_METHOD

METHOD PUBLIC getData : BOOL
VAR_INPUT
	par:INT;
END_VAR
CASE par OF
	0:
		getData:=getScrew();
	1:
		getData:=getEquip();
	2:
		getData:=getSteel();
	3:
		getData:=getSupport();		
ELSE
	getData:=FALSE;
END_CASE
END_METHOD

METHOD getSupport : BOOL
VAR_INPUT
END_VAR
	Support := arSupports[idxArSupport] ;
END_METHOD

METHOD PUBLIC AddSupport : BOOL
VAR_INPUT
END_VAR
VAR
	i,idxFind:INT:=0;
	step:UINT;
END_VAR

FOR i:=0 TO SIZE_SUPPORT DO
	IF arSupports[i].name = Support.name THEN
		AddSupport:=FALSE;
		RETURN;	
	END_IF	
END_FOR

FOR i:=1 TO SIZE_SUPPORT DO
		IF arSupports[i].name = "" THEN
			idxArSupport := i;
			arSupports[idxArSupport] := Support;
			AddSupport :=TRUE;
			RETURN;
		END_IF	
END_FOR

AddSupport :=FALSE;
END_METHOD

METHOD PUBLIC findName : BOOL
VAR_INPUT
	arr:POINTER TO dataBase;
	idxArr: UINT;
	step:uint;
	name: WSTRING;
END_VAR

VAR
	i:UINT:=0;
	step1:UINT:=156;
	arr1:POINTER TO dataBase;
	q: dataBase;
END_VAR
//сортировка массива имен файлов рецепта 

//так не работает 
	//  FOR i:=0 TO UINT_TO_INT(idxArr) BY UINT_TO_INT(step) DO 
	// 	 IF arr[i].name = name THEN// если текущая ячейка пуста, то переносим имя из последующей ячейки. Для исключения пробелов в списке
	// 		 idxFind:=i;
	// 		 findName:=TRUE;
	// 		 RETURN;
	// 	 END_IF	 
	//  END_FOR
	//  
	//   findName:=FALSE;
	//   idxFind:=0;
	
//	
i:=0;
WHILE NOT (findName OR i> idxArr) DO
	arr1:= arr+i;
	q:=arr1^;
	 IF q.name = name THEN// если текущая ячейка пуста, то переносим имя из последующей ячейки. Для исключения пробелов в списке
 		 findName:=TRUE;
	 END_IF	 
	 i:=i+step;
END_WHILE
END_METHOD

METHOD setSupport : BOOL
VAR_INPUT
END_VAR
 arSupports[idxArSupport] := Support;
END_METHOD

METHOD getEquip : BOOL
VAR_INPUT
END_VAR
	Equip := arEquip[idxArEquip] ;
END_METHOD

METHOD addSteel : BOOL
VAR_INPUT
END_VAR
VAR
	i,idxFind:INT:=0;
	step:UINT;
END_VAR
step:=SIZEOF(steel);

IF findName(ADR(arSteel), SIZE_SCREWS*step, step, Steel.name) THEN	
	AddSteel:=FALSE;
	RETURN;		
ELSE	
	FOR i:=0 TO SIZE_STEELS DO
		IF arSteel[i].name = "" THEN
			idxArSteel := i;
			arSteel[idxArSteel] := Steel;
			AddSteel :=TRUE;
			RETURN;
		END_IF	
	END_FOR
		AddSteel :=FALSE;

END_IF
END_METHOD

METHOD setEquip : BOOL
VAR_INPUT
END_VAR
	arEquip[idxArEquip]:= Equip;
END_METHOD

METHOD DelSupport : BOOL
VAR_INPUT
END_VAR
VAR
	i:int:=0;
END_VAR
VAR CONSTANT
	NOTHING :SupportType:=(arLength:=[0,0], name :="");
END_VAR
FOR i:=idxArSupport TO SIZE_SUPPORT DO 
	arSupports[i]:=arSupports[i+1];
	arSupports[i+1]:=NOTHING;
END_FOR
Support := NOTHING;
DelSupport:=TRUE;
END_METHOD

METHOD getScrew : BOOL
VAR_INPUT
END_VAR
	screw := arScrew[idxArScrew] ;
END_METHOD

METHOD setSteel : BOOL
VAR_INPUT
END_VAR
	arSteel[idxArSteel]:= Steel;
END_METHOD

END_PROGRAM

// Device/Application/POUs/gp/Actuators
PROGRAM Actuators
VAR_INPUT
	bCalibrateMode :BOOL;//режим калибровки линейки движения актуаторов
	bManualMode :BOOL;//режим ручного управления актуаторам
	bBtnStart	: BOOL; //запуск цикла в авто
	bBtnStop :BOOL;//импульс на выполнение задания	
	
	bDirRotate :BOOL;//направление вращение заготовки
	iCycleNumb	: INT;//число циклов
	iCalcStep 	: INT;//шаг смещения
	iStartPos :ARRAY [0..1] OF INT;//начальная поз. акт
	support :ARRAY [0..1] OF SupportType2;
END_VAR

VAR_OUTPUT
	iStage :INT;//стадия в режиме цикла 0-откл.; 1-инициал.; 2-стартовая; 3-цикл	
	iCycleCnt :INT;//кол-во циклов
	bActuatorsStop :BOOL;	
END_VAR

VAR
	bEn:BOOL;
	bActuatorsEnable :BOOL;

	iDr1_Cnt	: INT;
	iDr2_Cnt	: INT;

	bDr1_zero	: BOOL; //точка 0 актуатора 1
	bDr2_zero	: BOOL; //точка 0 актуатора 2	
	bDr1_worked	: BOOL; //работа актуатора 1 закончена
	bDr2_worked	: BOOL; //работа актуатора 2 закончена
	bDr1_error	: BOOL; //ошибка драйвера 1 дв1
	bDr2_error	: BOOL;	//ошибка драйвера 2 дв2
	bDr1_enable	: BOOL; //дв.1 включен
	bDr2_enable	: BOOL;	//дв.2 включен
	bDr1_Direct	: BOOL; //дв.1 направение
	bDr2_Direct	: BOOL;	//дв.2 направение
	bDr1_Impuls	: BOOL; //дв.1 генератор импульсов
	bDr2_Impuls	: BOOL;	//дв.2 генератор импульсов		
	bActuatorsStartByPR : BOOL;
	bCycleStop: BOOL;
	fbAct1,fbAct2 :fbActuator;
	 rImp1:R_TRIG;
	
	iDr1_startPos :INT;//начальная поз. акт 1	
	iDr2_startPos :INT;//начальная поз. акт 2
	
	iCurLenSuport1 :INT;
 	iCurLenSuport2 :INT;
END_VAR

	iDr1_startPos := iStartPos[0];//начальная поз. акт 1	
	iDr2_startPos := iStartPos[1];//начальная поз. акт 2

bCycleStop := iStage <> 0 AND ((iDr1_startPos > Sp.iMaxActuatorsMove OR iDr2_startPos > Sp.iMaxActuatorsMove ) OR 
bCalibrateMode OR bManualMode OR bBtnStop);


IF bCycleStop THEN
	iStage :=4;
	
ELSIF bBtnStart THEN
	iStage :=1;
	iCycleCnt:=0;	
END_IF
	
CASE iStage OF
	0://0-откл. 
		;
	
	1://1-инициал. 
		bActuatorsStop :=FALSE;
		
		fbAct1.iMode := fbAct2.iMode := 1;
		fbAct1.bBtnfrd := fbAct2.bBtnfrd := FALSE;
		fbAct1.bBtnbk:= NOT bDr1_zero; 
		fbAct2.bBtnbk:= NOT bDr2_zero;
		IF bDr1_zero AND bDr2_zero THEN
			iStage :=2;
		END_IF
		
	2://2-стартовая;
		fbAct1.bBtnbk := fbAct2.bBtnbk := FALSE;
		fbAct1.iMode := fbAct2.iMode := 2;
		fbAct1.iSetp := iDr1_startPos;  
		fbAct2.iSetp := iDr2_startPos;
		fbAct1.bBtnStart := fbAct2.bBtnStart := TRUE;
		
		IF NOT (fbAct1.bStart OR fbAct2.bStart) THEN
			fbAct1.bBtnStart := fbAct2.bBtnStart := FALSE;
			bActuatorsStop :=TRUE;
			iStage :=3;
		END_IF
		
	3:// 3-цикл	
		fbAct1.iMode := fbAct2.iMode := 3;
		fbAct1.iSetp :=	fbAct2.iSetp := iCalcStep;  
		
		rImp1(CLK:= bDr1_worked AND bDr2_worked);
		
		fbAct1.bBtnStart := fbAct2.bBtnStart := rImp1.Q;
		IF rImp1.Q THEN
			iCycleCnt := iCycleCnt +1;
		END_IF
		
		IF iCycleNumb < iCycleCnt THEN
			iStage :=4;
		END_IF
		
	4://откл
		fbAct1.bBtnbk := fbAct2.bBtnbk := FALSE;
		fbAct1.bBtnfrd := fbAct2.bBtnfrd := FALSE;
		fbAct1.bBtnStart := fbAct2.bBtnStart:= FALSE;
		fbAct1.iMode := fbAct2.iMode := 0;
			iStage :=0;
	
END_CASE
	
IF bManualMode THEN
	fbAct1.iMode:=fbAct2.iMode:=2;
ELSIF bCalibrateMode THEN
	fbAct1.iMode:=fbAct2.iMode:=1;
END_IF	


//установка крайнего положения актуатора по импульсам
	fbAct1(	iMode:= , 
			bBtnStart:= , 
			bZero:= bDr1_Zero, 
			bWorked:= bDr1_worked, 
			iCurCnt:= iDr1_Cnt,
			L_MAX:=sp.iMaxActuatorsMove, 
			iCurLength=> , 
			bStart=> , 
			iImpSetp=> , 
			bBk=> , 
			bFrd=> , 
			iMaxImp:= sp.iMaxImpDr1);
		
	fbAct2(	iMode:= , 
			bBtnStart:= , 
			bZero:= bDr2_zero, 
			bWorked:= bDr2_worked, 
			iCurCnt:= iDr2_Cnt, 
			L_MAX:=sp.iMaxActuatorsMove, 
			iCurLength=> , 
			bStart=> , 
			iImpSetp=> , 
			bBk=> , 
			bFrd=> , 
			iMaxImp:= sp.iMaxImpDr2 );
			
	IF support[0].bPosition THEN		
		iCurLenSuport1:= sp.iHeightMatrix + (support[0].arLength[1] - fbAct1.iCurLength);	
	ELSE
		iCurLenSuport1:= sp.iHeightMatrix + (support[0].arLength[0] - fbAct1.iCurLength);
	END_IF
		
	IF support[1].bPosition THEN		
		iCurLenSuport2:= sp.iHeightMatrix + (support[1].arLength[1] - fbAct2.iCurLength);	
	ELSE
		iCurLenSuport2:= sp.iHeightMatrix + (support[1].arLength[0] - fbAct2.iCurLength);
	END_IF		
	
	act_input();

ACTION ACT_INPUT:
	bDr1_error := DI1.6;//ошибка драйвера 1 дв1
	bDr2_error := DI1.7;//ошибка дравера 2 дв2
	bDr1_zero := DI1.8;//точка 0 актуатора 1
	bDr2_zero := DI1.9;//точка 0 актуатора 2	
	
	bDr1_enable	:= DO1.3;//вкл. драйвер 1
	bDr2_enable	:= DO1.4;//вкл. драйвер 2
	bDr1_Direct := DO1.5;//смена направления драйвера 1
	bDr2_Direct := DO1.6;//смена направления драйвера 2
	bDr1_Impuls := DO1.7;//шаговый импульс драйвера 1
	bDr2_Impuls := DO1.8;//	шаговый импульс драйвера 2	
	
	writeData.1 := bActuatorsEnable;//режим работы с актуаторами в автомате
	writeData.2 := fbAct1.bfrd;//актуатор 1 вперед
	writeData.3 := fbAct1.bBk;//актуатор 1 назад
	writeData.4 := fbAct2.bfrd;//актуатор 2 вперед
	writeData.5 := fbAct2.bBk;//актуатор 2 назад
	writeData.6 := bCalibrateMode;//актуатор 2 назад
	writeData.7 := bDr1_worked; //fbAct1.bStart;//
	writeData.8 := fbAct2.bStart;//
	writeData.9 := bActuatorsStop;// 
	
	writeImpMaxDr1 := sp.iMaxImpDr1;//максимальное число импульсов для шаговых дв
	writeImpMaxDr2 := sp.iMaxImpDr2;
	writeImpSetpDr1 := fbAct1.iImpSetp;//уставка импульсов на шаг в авто режиме
	writeImpSetpDr2 := fbAct2.iImpSetp;//уставка импульсов на шаг в авто режиме
	
	
	// := readStateDr.0;//работа актуатора 1 закончена
	//bDr2_worked := readStateDr.1;//работа актуатора 2 закончена
	bActuatorsStartByPR := readStateDr.2;//запуск в авто 
	
	iDr1_Cnt := readCntImpDr1;//текущее количество импульсов на дв. 1
	iDr2_Cnt := readCntImpDr2;//текущее количество импульсов на дв. 2
END_ACTION

END_PROGRAM

// Device/Application/POUs/gp/fbActuator
FUNCTION_BLOCK fbActuator
VAR_INPUT
	iMode :INT; //0-откл., 1-упр. с кнопок, 2-задание напрямую, мм, 3-авто, убывающий шаг, мм
	bCalibrate :BOOL;//сохранение крайней макс позиции актуатора
	bBtnBk :BOOL;//кн управления
	bBtnFrd :BOOL;//кн управления
	bBtnStart :BOOL;//импульс на выполнение задания

	bZero :BOOL;//крайняя нулевая позиция актуатора
	bWorked :BOOL;//актуатор выполнил задание
	iSetp :INT;// задание длины перемещения в мм
	iCurCnt :INT;//текущее значение счетчика импл. двиг. актуатора
	L_MAX : INT := 180; //максимальный ход актуаторов
END_VAR
VAR_OUTPUT
	iCurLength : INT;//положение актуатора в мм
	bStart :BOOL;//сигнал выполнение задания
	iImpSetp : INT; //значение шага в автоматическом режиме
	bBk :BOOL;//кн управления
	bFrd :BOOL;//кн управления
END_VAR
VAR
	iOldAccept :BOOL;
	iOldSetp :INT;
	tempImp :INT;
	iImpByMm :INT;
	rImpl :R_TRIG;
END_VAR

VAR_IN_OUT
	iMaxImp	: INT;
END_VAR

VAR CONSTANT
	
END_VAR

//установка крайнего положения актуатора по импульсам
IF bCalibrate AND NOT bZero AND iCurCnt > 0 THEN 
	iMaxImp := iCurCnt;	
END_IF

IF (iMaxImp / L_MAX) = 0 THEN
	iImpByMm:= 1 ;
ELSE
	iImpByMm:=(iMaxImp / L_MAX);
END_IF

iCurLength := iCurCnt*iImpByMm;
rImpl(CLK:= bBtnStart);

(*Данная конструкция нужна что бы сигнал потверждения bWorked успел обновится из за задержки обмена данных м/у устройсвтвами*)		
	IF iOldSetp <> iSetp AND NOT bWorked THEN
		iOldAccept :=FALSE;
		iOldSetp := iSetp;
	END_IF
	
	IF NOT iOldAccept THEN
		iOldAccept := bWorked;
	END_IF



CASE iMode OF
	1://1-упр. с кнопок,
		bBk := bBtnBk;//кн управления
		bFrd := bBtnFrd;//кн управления
	2:// 2-задание напрямую, мм,
		iImpSetp := iOldSetp/iImpByMm;	
		IF rImpl.Q THEN
			bStart := TRUE  ;
		ELSIF iOldAccept THEN
			bStart := FALSE  ;
		END_IF
		
		bBk := FALSE;//кн управления
		bFrd := FALSE;//кн управления
		
	3:// 3-авто, убывающий шаг, мм
		IF rImpl.Q THEN//перерасчет смещения актуаторов с новым циклом
			tempImp := iCurCnt - (iOldSetp/iImpByMm);
			IF tempImp >= 0 AND NOT bZero THEN // проверка на то что бы актуаторы не съехали за допустимый край
				iImpSetp := tempImp;	
			ELSE		
				iImpSetp := 0;
			END_IF
			bStart :=TRUE;
		ELSIF iOldAccept THEN
			bStart := FALSE  ;
		END_IF
		
		bBk := FALSE;//кн управления
		bFrd := FALSE;//кн управления
		
ELSE
	bStart := FALSE  ;
	bBk := FALSE;//кн управления
	bFrd := FALSE;//кн управления
END_CASE

END_FUNCTION_BLOCK

// Device/Application/POUs/_System/MessageEx
//Блок генерации дискретной аварии
FUNCTION_BLOCK MessageEx
VAR_INPUT
	bDI: BOOL;				(*контролируемый сигнал: 0 - авария, 1 - норма*)
	bEnbl: BOOL;				(*разрешение работы блока*)
	bLock: BOOL;				(*блокирование аварийного состояния до принудительного снятия 0 - не блок, 1 - блок*)
	iDelEn: INT;			(*задержка на появление сигнала*)
	bReset: BOOL;			(*сигнал сброса аварии*)
END_VAR
VAR_OUTPUT
	bOUT: BOOL;		(*состояние аварии: 0 - норма, 1 - авария*)
END_VAR
VAR
	fbDelay: TON;			(*TON для задержки на включение*)
	bErActive: BOOL;
END_VAR

IF bEnbl THEN
	fbDelay(IN:= NOT bDI, PT:= INT_TO_TIME(iDelEn)*1000, Q=> bErActive, ET=> );
ELSE 
	bErActive:=FALSE;	
END_IF

IF bErActive THEN 
	bOut:=TRUE;
ELSIF (bReset OR NOT bLock) AND_THEN NOT bErActive THEN
	bOut:=FALSE;
END_IF

END_FUNCTION_BLOCK

// Device/Application/POUs/gp/Operating_time_v1
FUNCTION_BLOCK Operating_time_v1
VAR_INPUT
	bEn:BOOL;
	iTimeTO : INT;
	bResetTO :	BOOL;
	bReset	:	BOOL;
END_VAR

VAR_IN_OUT
	op:OperTime;

END_VAR

VAR_OUTPUT
	bService :BOOL;
END_VAR
VAR
	bOn:	BOOL;
	minute	:TON;
	testref : BOOL := FALSE;
END_VAR

testref := __ISVALIDREF(op);

IF testref THEN 
	minute(In:= bOn, PT:=T#60s);
	
	IF minute.Q THEN
		op.dwTimeTotal := op.dwTimeTotal +1;
		op.dwMinTotal := op.dwMinTotal +1;
		op.dwMinSeans := op.dwMinSeans +1;
		
		IF op.dwMinTotal	=	60	THEN
			op.dwHourTotal	:=	op.dwHourTotal+1;
			op.dwHourSeans := op.dwHourSeans +1;
			op.dwMinSeans := op.dwMinTotal:=0;
		END_IF
		
	ELSIF bReset THEN
		op.dwHourTotal	:= op.dwMinTotal:=0;
	END_IF
	
	bOn:= bEn AND NOT minute.Q;
	
	IF NOT bEn THEN
		op.dwHourSeans := op.dwMinSeans :=0;
	END_IF
END_IF


IF (op.dwLastServ + INT_TO_DWORD(iTimeTO)) <= op.dwHourTotal THEN
	bService:=TRUE;
ELSIF bResetTO AND bService THEN
	op.dwLastServ := op.dwHourTotal;
	bService:=FALSE;
END_IF

END_FUNCTION_BLOCK

// Device/Application/POUs/gp/fbControl_sys
FUNCTION_BLOCK fbControl_sys
VAR_INPUT
	rCurLength	:	REAL;//текущее расстояние
	setX :recType2;//установленые значения точек в ручную
	recX :recType2;//установленые значения точек из рецептов
	rAccuracy	: REAL:=1.0; //относительная погрешность на движение мм
	bMoveFrd	: BOOL;//движение вперед в п-авто и ручном
	bMoveRev	: BOOL;//движение назад в п-авто и ручном		
	bReset:BOOL;//сброс ошибки 
	iTimeErr:	INT;//период м/у имп. энк. до аварии,c
	Accept :  Accept_struct;//принять данные
END_VAR

VAR_OUTPUT	
	rLengthFromX0 : REAL; //растояния от точки 0
	rCalcX2 : REAL;	//расчетная координата х2 относительно 0 на датчике
	rCalcX1 : REAL;	//расчетная координата х1 относительно 0 на датчике
	curX :recType2;	//текущее значение точек
	bAlarm:	BOOL;	//	Авария движ
	bNotX0:	BOOL;	//не установлен х0
END_VAR

VAR
	rSetLength : REAL;	//рабочая координата движения
	stage:INT:=0;
	mode0Stage:INT:=0;
	bVectorRev,bVectorFrd:bool;
	fbAlarms:	fbAlrmMove;	//
	nullX :recType2;
	
	bUpdate:BOOL;//обновить значения
END_VAR
VAR_TEMP						

												
END_VAR	
					
VAR CONSTANT

END_VAR

//nullX.rPosX0:=CurX.rPosX0;
//nullX.rPosX1:=CurX.rPosX1;
//nullX.rPosX2:=CurX.rPosX2;

//установка точeк
CASE iMode OF
	2: // ручной режимы
	//принияли стартовую точку исходя из текущего положения   
	 CurX.rPosX0 := rCurLength;			
	//обновить расчетные значения х0-х2	
		bUpdate	:= TRUE; 
ELSE
	//принияли стартовую точку из введеного числа   
	IF Accept.bX0 THEN   
		CurX.rPosX0 :=  setX.rPosX0;	
	ELSIF Accept.bX1 THEN
		CurX.rPosX1 := setX.rPosX1;	
	ELSIF Accept.bX2 THEN	
		//CurX := nullX;	
		CurX.rPosX2 := setX.rPosX2;
	ELSIF Accept.bRec THEN 
		CurX := recX;	
	END_IF
	//обновить расчетные значения х0-х2	
		bUpdate	:= Accept.bRec OR Accept.bX2 OR Accept.bX1 OR Accept.bX0; 
END_CASE;		
	
rLengthFromX0 := rCurLength - CurX.rPosX0;

IF	CurX.rPosX0	<> 0 THEN	//установлена точка х0
	IF	bUpdate THEN
		rCalcX1:= ((CurX.rPosX0+CurX.rPosX2)-CurX.rPosX1)+rAccuracy; //расчет х1 на линейки
		rCalcX2:= (CurX.rPosX0+CurX.rPosX2)-rAccuracy; //расчет х2 на линейки
		IF rCalcX2 <= rCalcX1 THEN//проверка на правильность х2 больше чем х1
			rCalcX1 := rCalcX2 - 1;
		END_IF		
	END_IF		
	bNotX0:=FALSE;
ELSE
	bNotX0:=TRUE;	
END_IF 

//блок анализа аварийных ситуаций
	fbAlarms(rLength:= rCurLength, 
			bStart:= (bMoveFrd OR bMoveRev), 
			iTimeErr:= iTimeErr, 
			bReset:= bReset, 
			bError=> bAlarm);			

//часть для актуаторов
 IF Accept.bAct THEN
	 CurX.iActuatorsMove :=  setX.iActuatorsMove;	
	 CurX.iActuatorsStartPos :=  setX.iActuatorsStartPos;	
	 CurX.iActuatorsStep :=  setX.iActuatorsStep;	
	 CurX.iCountCycle :=  setX.iCountCycle;	
	 CurX.bDirRotate :=  setX.bDirRotate;	
 END_IF
 
 IF Accept.bSup THEN
	CurX.support := setX.support;	
 END_IF

END_FUNCTION_BLOCK

// Device/Application/POUs/gp/fbAlrmMove
FUNCTION_BLOCK fbAlrmMove
VAR_INPUT
	rLength:	REAL;	//	текущая длина
	bStart:	BOOL;//	сигнал на движ 
	iTimeErr:INT;//уставка выдержки, с
	bReset:BOOL;// сброс ошиобки
END_VAR

VAR_OUTPUT
	bError:BOOL;//ошибка движения
END_VAR

VAR
	timerEr1:	TON;
	timerEr2:	TON;
	timerPeriod:	TON;
	rMemory:	REAL;	
	
END_VAR

VAR_TEMP
  	_time:	TIME;							
END_VAR

_time:=INT_TO_TIME(iTimeErr)*1000;

timerPeriod(in:=  NOT timerPeriod.Q, pt:=T#500MS);
	
IF timerPeriod.Q THEN
    rMemory := rLength;
END_IF;

timerEr1(IN := bStart AND rLength = rMemory,//если есть сигнал на дв. но нет перемещения
          PT:=_time);//Запускает аварийный таймер при начале движения

timerEr2(IN := NOT bStart AND (rLength <> rMemory),//если есть сигнал на дв. но нет перемещения
          PT:=_time);//Запускает аварийный таймер при начале движения
		  
IF timerEr1.Q  OR timerEr2.Q THEN
	bError := TRUE;
ELSIF bReset AND NOT timerEr1.Q AND NOT timerEr2.Q THEN
	bError := FALSE;
END_IF;

END_FUNCTION_BLOCK

// Device/Application/POUs/gp/simulateMove
FUNCTION_BLOCK simulateMove
VAR_INPUT
	frd:BOOL;
	rev:BOOL;
END_VAR
VAR_OUTPUT
	length:REAL:=0;
END_VAR
VAR
	delay:ton;
END_VAR

delay(in:= (frd OR rev) AND NOT delay.Q, pt:= T#400MS );

IF delay.Q AND frd AND NOT rev THEN
	length :=length+1;
ELSIF delay.Q AND rev AND NOT frd THEN
	length :=length-1;
END_IF

END_FUNCTION_BLOCK

// Device/Application/POUs/_System/WhatTime
FUNCTION WhatTime : bool
VAR_INPUT
END_VAR
VAR
	i:IDateTimeProvider;
	uliDateTime:ULINT;
END_VAR
VAR_OUTPUT
	uiSec:UINT;
	uiMsec:UINT;
END_VAR

uliDateTime:= util.GetDateTime();
util.SplitDateTime(uliDateTime:=uliDateTime,uiSecond=>uiSec,uiMilliseconds=>uiMsec);

END_FUNCTION

// Device/Application/POUs/_System/TimeSetup/TimeSetup
PROGRAM TimeSetup
VAR
	(*Часы реального времени*)
	m_RTC:RealTimeClock4;
	w_str_time:WSTRING;	
	w_str_dateM:WSTRING;
END_VAR

m_RTC(
	lang:= 'ru',
	Set_Year:= , 
	Set_Month:= , 
	Set_Day:= , 
	Set_Hour:= , 
	Set_Minute:= , 
	Set_Second:= , 
	Add_Year:= , 
	Add_Month:= , 
	Add_Day:= , 
	Add_Hour:= , 
	Add_Minute:= , 
	Add_Second:= , 
	Sub_Year:= , 
	Sub_Month:= , 
	Sub_Day:= , 
	Sub_Hour:= , 
	Sub_Minute:= , 
	Sub_Second:= , 
	RTC=> , 
	Year=> , 
	Month=> , 
	Day=> , 
	Hour=> , 
	Minute=> , 
	Second=> , 
	w_str_time=> w_str_time, 
	w_str_dateM=> w_str_dateM);

END_PROGRAM

// Device/Application/POUs/_System/TimeSetup/RealTimeClock4
FUNCTION_BLOCK RealTimeClock4
VAR_INPUT
	Lang:			STRING;
	Set_Year:		 UINT;
	Set_Month:		 UINT;
	Set_Day:		 Uint;
	Set_Hour:		 Uint;
	Set_Minute:		 Uint;
	Set_Second:		 UINT;	
	Add_Year:		 BOOL;
	Add_Month:		 BOOL;
	Add_Day:		 BOOL;
	Add_Hour:		 BOOL;
	Add_Minute:		 BOOL;
	Add_Second:		 BOOL;
	Sub_Year:		 BOOL;
	Sub_Month:		 BOOL;
	Sub_Day:		 BOOL;
	Sub_Hour:		 BOOL;
	Sub_Minute:		 BOOL;
	Sub_Second:		 BOOL;
END_VAR

VAR_OUTPUT
	RTC:		 DT;
	Year:		 UINT;
	Month:		 UINT;
	Day:		 UINT;
	Hour:		 UINT;
	Minute:		 UINT;
	Second:		 UINT;
	w_str_time:		WSTRING;	(*Получаем Время в виде строки - статичное изображение*)                 
	w_str_dateM:	WSTRING;	(*Получаем Дату в виде строки - месяц буквами*)
END_VAR
VAR
	GetTime: DTU.GetDateAndTime;
	SetTime: DTU.SetDateAndTime;
	RT_TIME:R_TRIG;
	RT_Add_Year:		 R_TRIG;
	RT_Add_Month:		 R_TRIG;
	RT_Add_Day:			 R_TRIG;
	RT_Add_Hour:		 R_TRIG;
	RT_Add_Minute:		 R_TRIG;
	RT_Add_Second:		 R_TRIG;
	RT_Sub_Year:		 R_TRIG;
	RT_Sub_Month:		 R_TRIG;
	RT_Sub_Day:			 R_TRIG;
	RT_Sub_Hour:		 R_TRIG;
	RT_Sub_Minute:		 R_TRIG;
	RT_Sub_Second:		 R_TRIG;
	Error: DTU.ERROR;
	Set:BOOL;
	
	Update_Year:		 UpdateUint;
	Update_Month:		 UpdateUint;
	Update_Day:		 	UpdateUint;
	Update_Hour:		 UpdateUint;
	Update_Minute:		 UpdateUint;
	Update_Second:		 UpdateUint;
	
	(*Расчет високосного года*)
	leap_year: BOOL;
	x1:WORD;
	x2:WORD;
	x3:WORD;
	(*последний день текущего месяца*)
	EndDay: UINT;
	(*конвертируем дату и время в текст*)
	Second_old:UINT;
	MonthWS:WSTRING;
END_VAR

(*Получаем системное время в формате DATE_AND_TIME*)
GetTime(xExecute:= NOT(GetTime.xDone));
RT_TIME(CLK:=GetTime.xDone);
IF RT_TIME.Q AND GetTime.xBusy=FALSE AND GetTime.xError=FALSE AND GetTime.eError=0 THEN
	RTC:=GetTime.dtDateAndTime;
	(*Разбираем системное время*)
	Error:=DTU.DTSplit(
			dtDateAndTime:= RTC, 
			puiYear:= ADR(Year), 
			puiMonth:= ADR(Month), 
			puiDay:= ADR(Day), 
			puiHour:= ADR(Hour), 
			puiMinute:= ADR(Minute), 
			puiSecond:= ADR(Second));
	(*Собираем время в строку*)	
END_IF



	IF Second_old<>Second THEN
		w_str_time:=wconcat(WORD_TO_WSTRING(Hour)," : ");
		IF Minute < 10
		THEN
			w_str_time:=wconcat(w_str_time,"0");
		END_IF;	
		w_str_time:=wconcat(w_str_time,WORD_TO_WSTRING(Minute));			
		w_str_time:=wconcat(w_str_time," : ");
		IF Second < 10
		THEN
			w_str_time:=wconcat(w_str_time,"0");
		END_IF;	
		w_str_time:=wconcat(w_str_time,WORD_TO_WSTRING(Second));			
		
		IF 	Lang='ru' THEN	
			CASE Month OF
				1:
					MonthWS:="января";
				2:
					MonthWS:="февраля";		
				3:
					MonthWS:="марта";		
				4:
					MonthWS:="апреля";		
				5:
					MonthWS:="мая";		
				6:
					MonthWS:="июня";		
				7:
					MonthWS:="июля";		
				8:
					MonthWS:="августа";		
				9:
					MonthWS:="сентября";		
				10:
					MonthWS:="октября";		
				11:
					MonthWS:="ноября";		
				12:
					MonthWS:="декабря";		
			END_CASE
		ELSE
			CASE Month OF
				1:
					MonthWS:="January";
				2:
					MonthWS:="February";		
				3:
					MonthWS:="March";		
				4:
					MonthWS:="April";		
				5:
					MonthWS:="May";		
				6:
					MonthWS:="June";		
				7:
					MonthWS:="July";		
				8:
					MonthWS:="August";		
				9:
					MonthWS:="September";		
				10:
					MonthWS:="October";		
				11:
					MonthWS:="November";		
				12:
					MonthWS:="December";		
			END_CASE
		END_IF
		

		IF Lang='ru' THEN	
			w_str_dateM:=wconcat(WORD_TO_WSTRING(Day)," ");
			w_str_dateM:=wconcat(w_str_dateM,MonthWS);
			w_str_dateM:=wconcat(w_str_dateM," ");
			w_str_dateM:=wconcat(w_str_dateM,WORD_TO_WSTRING(Year));
			w_str_dateM:=wconcat(w_str_dateM,"г.");
		ELSE
			w_str_dateM:=wconcat(MonthWS," ");
			w_str_dateM:=wconcat(w_str_dateM,WORD_TO_WSTRING(Day));
			w_str_dateM:=wconcat(w_str_dateM,"th, ");
			w_str_dateM:=wconcat(w_str_dateM,WORD_TO_WSTRING(Year));
		END_IF
	END_IF
	
Second_old:=Second;


(*Определяем високосный год или нет*)
x1:= Year MOD 4;
x2:= Year MOD 100;
x3:= Year MOD 400;

IF (x3=0) OR (x1=0 AND x2<>0 ) THEN
	leap_year:=TRUE;
END_IF

IF (x1<>0) OR (x2=0 AND x3<>0) THEN
	leap_year:=FALSE;
END_IF

(*Определяем последний день текущего месяца*)
CASE Month OF
	1:
		EndDay:=31;
	2:
		IF leap_year THEN
			EndDay:=29;
		ELSE
			EndDay:=28;
		END_IF
	3:
		EndDay:=31;
	4:
		EndDay:=30;
	5:
		EndDay:=31;
	6:
		EndDay:=30;
	7:
		EndDay:=31;
	8:
		EndDay:=31;
	9:
		EndDay:=30;
	10:
		EndDay:=31;
	11:
		EndDay:=30;
	12:
		EndDay:=31;	
END_CASE


(*Управление временем через логичские входы*)
RT_Add_Year		(	CLK:=Add_Year)	;
RT_Add_Month	(	CLK:=Add_Month)	;
RT_Add_Day		(	CLK:=Add_Day)	;
RT_Add_Hour		(	CLK:=Add_Hour)	;
RT_Add_Minute	(	CLK:=Add_Minute);	
RT_Add_Second	(	CLK:=Add_Second);	
RT_Sub_Year		(	CLK:=Sub_Year)	;  
RT_Sub_Month	(	CLK:=Sub_Month) ;
RT_Sub_Day		(	CLK:=Sub_Day)	;   
RT_Sub_Hour		(	CLK:=Sub_Hour)	;  
RT_Sub_Minute	(	CLK:=Sub_Minute);	
RT_Sub_Second	(	CLK:=Sub_Second);	


(*ГОД*)
IF RT_Add_Year.Q THEN
	Year:=Year+1;
	IF Year>2038 THEN
		Year:=2038;
	END_IF
END_IF

IF RT_Sub_Year.Q THEN
	Year:=Year-1;
	IF Year<1970 THEN
		Year:=1970;
	END_IF
END_IF


(*Месяц*)
IF RT_Add_Month.Q THEN
	Month:=Month+1;
	IF Month >12 AND Month<20 THEN
		Month:=1;	
	END_IF
END_IF

IF RT_Sub_Month.Q THEN
	Month:=Month-1;
	IF (Month <=65535 AND Month>65500) or Month=0 THEN
		Month:=12;	
	END_IF
END_IF


(*День*)
IF RT_Add_Day.Q THEN
	Day:=Day+1;
	IF Day >EndDay AND Day<40 THEN
		Day:=1;	
	END_IF
END_IF

IF RT_Sub_Day.Q THEN
	Day:=Day-1;
	IF (Day <=65535 AND Day>65500) OR Day=0 THEN
		Day:=EndDay;	
	END_IF
END_IF

(*Час*)
IF RT_Add_Hour.Q THEN
	Hour:=Hour+1;
	IF Hour >23 AND Hour<30 THEN
		Hour:=0;	
	END_IF
END_IF

IF RT_Sub_Hour.Q THEN
	Hour:=Hour-1;
	IF Hour <=65535 AND Hour>65500 THEN
		Hour:=23;	
	END_IF
END_IF


(*Минута*)
IF RT_Add_Minute.Q THEN
	Minute:=Minute+1;
	IF Minute >59 AND Minute<70 THEN
		Minute:=0;	
	END_IF
END_IF

IF RT_Sub_Minute.Q THEN
	Minute:=Minute-1;
	IF Minute <=65535 AND Minute>65500 THEN
		Minute:=59;	
	END_IF
END_IF

(*Секунда*)
IF RT_Add_Second.Q THEN
	Second:=Second+1;
	IF Second >59 AND Second<70 THEN
		Second:=0;	
	END_IF
END_IF

IF RT_Sub_Second.Q THEN
	Second:=Second-1;
	IF Second <=65535 AND Second>65500 THEN
		Second:=59;	
	END_IF
END_IF


(*Если введено новое значение*)
Update_Year(In:= Set_Year, Set=> );
Update_Month(In:= Set_Month, Set=> );
Update_Day(In:= Set_Day, Set=> );
Update_Hour(In:= Set_Hour, Set=> );
Update_Minute(In:= Set_Minute, Set=> );
Update_Second(In:= Set_Second, Set=> );

IF Update_Year.Set THEN
	(*Собираем системное время*)	
	RTC:=DTU.DTConcat(
		uiYear:= Set_Year, 
		uiMonth:= Month, 
		uiDay:= Day, 
		uiHour:= Hour, 
		uiMinute:= Minute, 
		uiSecond:= Second, 
		peError:= ADR(Error));
		Set:=TRUE;
END_IF

IF Update_Month.Set THEN
	(*Собираем системное время*)	
	RTC:=DTU.DTConcat(
		uiYear:= Year, 
		uiMonth:= Set_Month, 
		uiDay:= Day, 
		uiHour:= Hour, 
		uiMinute:= Minute, 
		uiSecond:= Second, 
		peError:= ADR(Error));
		Set:=TRUE;
END_IF

IF Update_Day.Set THEN
	(*Собираем системное время*)	
	RTC:=DTU.DTConcat(
		uiYear:= Year, 
		uiMonth:= Month, 
		uiDay:= Set_Day, 
		uiHour:= Hour, 
		uiMinute:= Minute, 
		uiSecond:= Second, 
		peError:= ADR(Error));
		Set:=TRUE;
END_IF

IF Update_Hour.Set THEN
	(*Собираем системное время*)	
	RTC:=DTU.DTConcat(
		uiYear:= Year, 
		uiMonth:= Month, 
		uiDay:= Day, 
		uiHour:= Set_Hour, 
		uiMinute:= Minute, 
		uiSecond:= Second, 
		peError:= ADR(Error));
		Set:=TRUE;
END_IF

IF Update_Minute.Set THEN
	(*Собираем системное время*)	
	RTC:=DTU.DTConcat(
		uiYear:= Year, 
		uiMonth:= Month, 
		uiDay:= Day, 
		uiHour:= Hour, 
		uiMinute:= Set_Minute, 
		uiSecond:= Second, 
		peError:= ADR(Error));
		Set:=TRUE;
END_IF

IF Update_Second.Set THEN
	(*Собираем системное время*)	
	RTC:=DTU.DTConcat(
		uiYear:= Year, 
		uiMonth:= Month, 
		uiDay:= Day, 
		uiHour:= Hour, 
		uiMinute:= Minute, 
		uiSecond:= Set_Second, 
		peError:= ADR(Error));
		Set:=TRUE;
END_IF


(*Пишем новое значение*)
IF	RT_Add_Year.Q OR RT_Add_Month.Q OR RT_Add_Day.Q OR RT_Add_Hour.Q OR RT_Add_Minute.Q OR RT_Add_Second.Q OR 
	RT_Sub_Year.Q OR RT_Sub_Month.Q OR RT_Sub_Day.Q OR RT_Sub_Hour.Q OR RT_Sub_Minute.Q OR RT_Sub_Second.Q THEN
	
	(*Собираем системное время*)	
	RTC:=DTU.DTConcat(
		uiYear:= Year, 
		uiMonth:= Month, 
		uiDay:= Day, 
		uiHour:= Hour, 
		uiMinute:= Minute, 
		uiSecond:= Second, 
		peError:= ADR(Error));
		Set:=TRUE;
END_IF

IF Set THEN
	SetTime(
		xExecute:= TRUE, 
		dtDateAndTime:= RTC, 
		xDone=> , 
		xBusy=> , 
		xError=> , 
		eError=> );
	
	IF SetTime.xDone  AND SetTime.xError=FALSE  THEN
		SetTime(xExecute:= FALSE);
		Set:=FALSE;
		sysexecute('/etc/rc.sync &');
	ELSE
		SetTime(xExecute:= FALSE);
	END_IF
END_IF

END_FUNCTION_BLOCK

// Device/Application/POUs/_System/TimeSetup/UpdateUint
FUNCTION_BLOCK UpdateUint
VAR_INPUT
	In: UINT;
END_VAR
VAR_OUTPUT
	Set: BOOL;
END_VAR
VAR
	In_OLD: UINT;
	rt:R_Trig;
END_VAR

rt(CLK:=IN<>IN_OLD);

Set:=rt.Q;

In_OLD:=IN;

END_FUNCTION_BLOCK

// Device/Application/POUs/_System/waitingScreen
FUNCTION_BLOCK waitingScreen
VAR_INPUT
	on:	BOOL; //включение анимации
	Xmin	:INT:=0; //граница экрана по Х
	Xmax	:INT:=600; //граница экрана по Х
	Ymin 	:INT:=-10;	//граница экрана по Y
	Ymax	:INT:=395; //граница экрана по Y
END_VAR
VAR_OUTPUT
	x	:INT; //координата перемещения х
	y	:INT; //координата перемещения y

END_VAR
VAR
	middle_x	:INT;
	middle_y	:INT;
	
	limMinY		:BOOL;
	limMaxY		:BOOL;
	
	limMinX		:BOOL;
	limMaxX		:BOOL;
	tonOffset	:TON;
END_VAR

middle_x:= (Xmax-Xmin)/2;
middle_y:= (Ymax-Ymin)/2;

	IF NOT on THEN 
		x:= middle_x;
		y:= middle_y;
		limMaxX :=limMaxY :=TRUE;
	END_IF;


	IF Xmax < x THEN 
		limMaxX :=TRUE;
		limMinX :=FALSE;
	ELSIF Xmin > x THEN
		limMaxX :=FALSE;
		limMinX :=TRUE;
	END_IF;
	
	IF Ymax < y THEN 
		limMaxY :=TRUE;
		limMinY :=FALSE;
	ELSIF Ymin > y THEN
		limMaxY :=FALSE;
		limMinY :=TRUE;
	END_IF;

 tonOffSet(In:= on AND NOT tonOffSet.Q ,PT:=T#1S);
	
IF tonOffSet.Q THEN
	IF limMinX THEN
		x:= x+3;
	ELSIF limMaxX THEN
		x:= x-3;
	END_IF;
	
	IF limMinY THEN
		y:= y+3;
	ELSIF limMaxY THEN
		y:= y-3;
	END_IF;
END_IF;

END_FUNCTION_BLOCK

// Device/Application/POUs/_System/TimeToString
FUNCTION_BLOCK TimeToString
VAR_INPUT
	in:OperTime;

END_VAR

VAR_OUTPUT
	wsDataSeans		:	WSTRING;	
	wsDataTotal		:	WSTRING;	
END_VAR

	wsDataSeans:=wconcat(DWORD_TO_WSTRING(in.dwHourSeans)," : ");
	IF in.dwMinSeans < 10
	THEN
		wsDataSeans:=wconcat(wsDataSeans,"0");
	END_IF;	
	wsDataSeans:=wconcat(wsDataSeans,DWORD_TO_WSTRING(in.dwMinSeans));
	
			
	wsDataTotal:=wconcat(DWORD_TO_WSTRING(in.dwHourTotal)," : ");
	IF in.dwMinTotal < 10
	THEN
		wsDataTotal:=wconcat(wsDataTotal,"0");
	END_IF;	
	wsDataTotal:=wconcat(wsDataTotal,DWORD_TO_WSTRING(in.dwMinTotal));

END_FUNCTION_BLOCK

// Device/Application/POUs/_System/ConvToVolt
FUNCTION_BLOCK ConvToVolt
VAR_INPUT
	rIn: REAL; 
	bMode: BOOL; //0 - вых.сигн 0..10В, 1 - вых.сигн 2..10В
END_VAR

VAR_OUTPUT
	wOut: WORD;
END_VAR
VAR
	TOV: RangeConvert;
END_VAR

VAR CONSTANT
    NULL : REAL := 0.0;
	FULL : REAL := 100.0;
    _10V : REAL := 1000.0;
	_2V : REAL := 200.0;
END_VAR

TOV(InVal := rIn, I1 := NULL, I2 := FULL, O1 := SEL(bMode, NULL, _2V), O2 := _10V, Lim := TRUE); // RangeConvert
wOut := SEL(NULL = rIn, REAL_TO_WORD(TOV.OutVal), 0);

END_FUNCTION_BLOCK

// Device/Application/POUs/_System/RangeConvert
FUNCTION_BLOCK RangeConvert
VAR_INPUT
	//Входной сигнал
   InVal:REAL;
   //мин. предел ВХОДН. сигнала
   I1:REAL;
   //мах. предел ВХОДН. сигнала
   I2:REAL;
   //мин. предел ВЫХОД. сигнала
   O1:REAL;
   //мах. предел ВЫХОД. сигнала
   O2:REAL;
   //вкл. контроль превышения пределов (если вых сигнал получится больше или меньше вых предела, то он будет приравненм к вых.пределу)
   Lim:BOOL;
END_VAR
VAR_OUTPUT
	//Выходной сигнал
   OutVal:REAL;
END_VAR
VAR
   delta_I:REAL;
   delta_O:REAL;
   koef:REAL;
END_VAR

delta_I:=I2-I1;
delta_O:=O2-O1;

IF delta_I = 0 THEN
  OutVal:=(O1+O2)/2;
  
ELSE
	  koef :=(InVal-I1)/delta_I;
	  OutVal :=O1+koef*delta_O;
	 
	 IF Lim THEN
	
			IF OutVal>O2 THEN
			 	OutVal:=O2;
			END_IF;
			
			IF OutVal<O1 THEN
			  	OutVal:=O1;
			END_IF;
	  END_IF;
END_IF;

END_FUNCTION_BLOCK

// Device/Application/POUs/_System/fcSortInt
FUNCTION fcSortInt : BOOL
VAR_INPUT
	arr	:POINTER TO INT;
	length: INT;//размер массива
END_VAR
VAR
	i,ii:INT;
	temp:INT;
END_VAR

//пузырьковая сортировка
FOR i:=0 TO length DO
	FOR ii:=1 TO length DO
		IF arr[i] < arr[ii] AND arr[i]<>0 THEN
			temp := arr[ii];
			arr[ii]:= arr[i];
			arr[i]:= temp;
		END_IF
	END_FOR
END_FOR

END_FUNCTION

// Device/Application/POUs/_System/TimeSetup/Day2weekDay
FUNCTION Day2weekDay : UINT
VAR_INPUT
	Year: UINT; 
	Month: UINT; 
	Day: UINT;
END_VAR
VAR
	a:UINT;
	y:UINT;
	m:UINT;
END_VAR

	a := 14 - Month;
	a := a/12;
 	y := year - a;
 	m := month + (12 * a) - 2;
 	Day2weekDay := (7000 + (day + y + (y / 4) - (y / 100) + (y / 400) + ((31 * m) / 12))) MOD 7;

END_FUNCTION

// Device/Application/POUs/_System/simpleSPAD
FUNCTION_BLOCK simpleSPAD
	//скидывает выходной сигнал от мах до мин, за время Т. по имп. от start
VAR_INPUT
	bStart	:BOOL; //начало спада
	bRes	:BOOL; //сбрасывает спад в мин по импл
	bMode	:BOOL; //0-спад. 1-подъем
	
	rMax	:REAL:=100.0; // начальное максимальное зн
	rMin	:REAL:=0.0; //минимальное конечное зн
	iT	:INT:=10;//время с
END_VAR
VAR_OUTPUT
	bActive :BOOL; //работа спада
	rOut	:REAL;

END_VAR
VAR
	r_start: R_TRIG;
	r_res: R_TRIG;
	rs_start:BOOL;

	tPeriod:TIME;
	ton:ton;
	
	dif: real;
END_VAR



r_start(CLK:=bStart);
r_res(CLK:=bRes);

IF r_start.Q THEN
	rs_start:=TRUE;
	IF NOT bMode THEN
		rOut:= rMax;
	ELSE 
		rOut :=rMin;
	END_IF;	
	
ELSIF NOT bStart THEN
	rs_start:=FALSE;
ELSIF r_res.Q THEN	
	rs_start:=FALSE;
	rOut :=rMin;
END_IF

dif:= (INT_TO_REAL(it)*1000)/(rMax-rMin);

tPeriod:= REAL_TO_TIME(dif);

bActive := rs_start AND ((bMode AND rOut<rMax) OR (NOT bMode AND rOut>rMin));
ton(IN:=bActive AND NOT ton.Q, pt := tPeriod);

IF ton.Q AND NOT bMode THEN
	rOut:= rOut-1;
ELSIF ton.Q AND bMode THEN
	rOut:= rOut+1;
END_IF

END_FUNCTION_BLOCK

// Device/Application/POUs/gp/fbSensor
FUNCTION_BLOCK fbSensor
VAR_INPUT
	rRawVal :REAL:=0.0; //вх.сигнал с датчика
	wRawStatus 	:WORD:=0; // вх. статус входного сигнала с датчика
	bOnConrolWarnLim:BOOL:=FALSE;//контроль предупредительных пределов
	bOnConrolErLim:BOOL:=FALSE;//контроль аварийных пределов
	rOffset			:	REAL	:=0; //Смещение показания датчика
	rH				:	REAL	:=5; //уставка вернего предупред предела
	rHH				:	REAL	:=251;//уставка вернего аварийного предела
	rL				:	REAL	:=240;//уставка нижнего предупред предела
	rLL				:	REAL	:=-1;//уставка нижнего авраийного предела	

	rMinValue		:	REAL	:= 0;	(*Минимум технологическое значение*)
	rMaxValue		:	REAL	:= 250;(*Максимум технологическое значение*)
	bReset	: BOOL;
END_VAR

VAR_OUTPUT
	rValue	:REAL;//Вых. значение с датчика
	iStat	:INT;//вых. 0-Норма; 1-Нижний предупредительный порог; 2-Верхний предупредительный порог; 3-Нижний аварийный порог;  4-Верхний аварийный порог; 5-авария датчика; 6-Режим блокировки сигнализации; 7-Ремонтный режим
	bError 	 	: 	BOOL;		//Общая ошибка
	bSnsErr		:BOOL:=FALSE;	//ошибка датчика
	bSnsH		:BOOL:=FALSE;	//ошибка верхнего предела
	bSnsHH		:BOOL:=FALSE;	//ошибка аварийного верхнего предела
	bSnsL		:BOOL:=FALSE;	//ошибка нижнего предела
	bSnsLL		:BOOL:=FALSE;	//ошибка аварийного нижнего предела
END_VAR
VAR
	Range: RangeConvert;
	MeX: MessageEx;
	MeXH					:	MessageEx;
	MeXHH					:	MessageEx;
	MeXL					:	MessageEx;
	MeXLL					:	MessageEx;
END_VAR


Range(InVal:= rRawVal, 
	I1:= 0, 
	I2:= 100, 
	O1:= rMinValue, 
	O2:= rMaxValue, 
	Lim:= TRUE, 
	OutVal=> );

	rValue := Range.OutVal + Sp.rOffset;

	MeX(bDI:= wRawStatus = 0,
		bEnbl:= TRUE,
		bLock:= TRUE ,
		iDelEn:=2,
		bReset:=bReset ,
		bOUT=> bSnsErr);

	IF NOT bSnsErr THEN
		IF  bOnConrolWarnLim THEN
			MeXH(bDI:=FALSE,
				bEnbl:= rValue >rH,
				bLock:= FALSE,
				iDelEn:=0,
				bReset:=bReset ,
				bOUT=> bSnsH);
				
			MeXL(bDI:=FALSE,
				bEnbl:= rValue < rL,
				bLock:= FALSE ,
				iDelEn:=0,
				bReset:=bReset ,
				bOUT=> bSnsL);
		END_IF
		IF  bOnConrolErLim THEN		
			MeXHH(bDI:= FALSE,
				bEnbl:= rValue > rHH,
				bLock:= TRUE ,
				iDelEn:=0,
				bReset:=bReset ,
				bOUT=> bSnsHH);
		
	
			MeXLL(bDI:= FALSE,
				bEnbl:= rValue  < rLL,
				bLock:= TRUE ,
				iDelEn:=0,
				bReset:=bReset ,
				bOUT=> bSnsLL);	
		END_IF
	ELSE
		bSnsH:=FALSE; bSnsHH :=FALSE; bSnsL:=FALSE; bSnsLL := FALSE;
	END_IF

bError := bSnsErr OR bSnsH OR bSnsHH OR bSnsL OR bSnsLL ;

(*0-Норма; 1-Нижний предупредительный порог; 3-Нижний аварийный порог; 2-Верхний предупредительный порог;  4-Верхний аварийный порог; 5-авария датчика; *)

	IF bSnsErr  THEN
		iStat :=5;
	ELSIF bSnsHH	 THEN
		iStat :=4;
	ELSIF bSnsH	THEN
		iStat :=3;
	ELSIF bSnsLL THEN
		iStat :=2;
	ELSIF bSnsL	 THEN
		iStat :=1;
	ELSE
		iStat :=0;
	END_IF

END_FUNCTION_BLOCK

// Device/Application/POUs/_System/getEquipKeypad
FUNCTION getEquipKeypad : WSTRING
VAR_INPUT
	sDirection: INT:=0;
	sTypeEquip:	INT:=0;
	sHeight:	WSTRING:="100";
	sAngle:	WSTRING:="10";
	sMidle:	wSTRING:="100";
END_VAR
VAR
	
END_VAR


getEquipKeypad:= WCONCAT(MUX(sDirection,"L","R"), WCONCAT("-",  WCONCAT(MUX(sTypeEquip,"N","F"), WCONCAT("-", 
					WCONCAT(sHeight, WCONCAT("-", WCONCAT(sAngle, WCONCAT("-", sMidle))))))));

END_FUNCTION

// Device/Application/POUs/_System/WhatCycleTime
FUNCTION WhatCycleTime : UINT
VAR_INPUT
	in:test;
END_VAR
VAR
END_VAR

WhatCycleTime:=(in.endCycle[0]*1000+in.endCycle[1]) - (in.startCycle[0]*1000+in.startCycle[1]);

END_FUNCTION

// Device/Application/POUs/_System/dword2real
FUNCTION dword2real : REAL
VAR_INPUT
	aWord		:	ARRAY [0..1] OF WORD;
END_VAR
VAR
	x			:	REAL;
	adress		:	POINTER TO WORD;
	adress2		:	POINTER TO WORD;
	i			:	INT;
END_VAR

adress2:=ADR(x);
adress2^:=aWord[1];
adress2:=adress2+2;	
adress2^:=aWord[0];
dword2real:=x;

END_FUNCTION

// Device/Application/POUs/gp/fbCylinder
FUNCTION_BLOCK fbCylinder
VAR_INPUT
	rCurLength	: REAL;//текущее расстояние
	rSetLength : REAL;//стартовая точка точка
	bMode	: BOOL;//0-дв. по коорд, 1-дв. по нажатию 
	bFrd	: BOOL;//движение вперед в п-авто и ручном
	bRev	: BOOL;//движение назад в п-авто и ручном	
	bStopFrd : BOOL;//крайняя точка движения вперед
	bStopRev : BOOL;//крайняя точка движения назад
	bReset:BOOL;//сброс ошибки 
	iTimeErr:	INT;//период м/у имп. энк. до аварии,c
END_VAR

VAR_OUTPUT	
	bMoveFrd:	BOOL;	//движение вперед
	bMoveRev:	BOOL;	//движение обратно
	bAlarm:	BOOL;	//	Авария движ
	iStatus:	INT	;//	0 - на месте, 1 - надо вперед, 2 - надо назад

END_VAR

VAR
	rDifference:	REAL;	
	fbAlarms:	fbAlrmMove;	//
	vector_frd:	BOOL;//	
	vector_rev: BOOL;//	
	rSaveLength:REAL;
END_VAR

VAR_IN_OUT
END_VAR

VAR_TEMP						

												
END_VAR	
					
VAR CONSTANT

END_VAR

//блок анализа аварийных ситуаций
	fbAlarms(rLength:= rCurLength, 
			bStart:= bMoveFrd OR bMoveRev, 
			iTimeErr:= iTimeErr, 
			bReset:= bReset, 
			bError=> bAlarm);			
	
IF (iStatus = 0 OR ABS(rSaveLength-rSetLength)> 1.0 ) AND rSaveLength<>rSetLength THEN	// определяем новую рабочую уставку
	rSaveLength := rSetLength;
	istatus:=1;
END_IF

rDifference := rSaveLength - rCurLength;

IF  bMode  THEN
	 vector_frd := bFrd;
	 vector_rev := bRev;
ELSE
	CASE iStatus OF 
		0://на месте 
				vector_rev := FALSE;
				vector_frd := FALSE;
		1:	
			//определяем направление движения
			IF rDifference < 0 THEN
				istatus:=3;			
			ELSIF rDifference >=  0 THEN
				istatus:=2;
			END_IF
	
		2: //надо вперед
				vector_rev := bRev;
				vector_frd := bFrd;
				
			IF  rSaveLength <= rCurLength THEN
				istatus:=0;
			END_IF						

		3: //надо назад
				vector_rev := bFrd OR bRev;	
				vector_frd := FALSE;
				
			IF  rSaveLength >= rCurLength THEN
				vector_rev := FALSE;
				istatus:=0;
			END_IF
	END_CASE;   
 END_IF

// вкл выходов
bMoveFrd:=	vector_frd AND NOT(bAlarm OR bStopFrd OR bMoveRev);
bMoveRev:=	vector_rev AND NOT(bAlarm OR bStopRev OR bMoveFrd);

END_FUNCTION_BLOCK

